Yaskawa INFORM job: X2_38-47,64(1)(90,180).JBI

/JOB
//NAME X2_38-47,64(1)(90,180)
//POS
///NPOS 477,477,477,26,0,0
///TOOL 0
///POSTYPE PULSE
///PULSE
C00000=10776,-116726,-133110,-1428,79202,-268
C00001=121301,-101656,-130574,15140,106953,26685
C00002=120740,-100574,-124017,14929,103680,26084
C00003=120691,-100743,-123189,14892,103111,25997
C00004=120691,-101012,-123023,14875,102879,25968
C00005=120694,-100727,-123199,14892,103125,25999
C00006=120263,-93974,-120700,15099,105066,26103
C00007=120694,-100727,-123199,14892,103125,25999
C00008=121303,-103883,-129892,15002,105440,26491
C00009=121309,-101301,-130428,15148,107041,26699
C00010=120755,-99767,-124232,14968,104207,26155
C00011=120700,-99774,-123449,14938,103747,26079
C00012=120700,-100712,-122892,14879,102948,25979
C00013=120685,-100384,-123078,14901,103225,26009
C00014=120255,-93653,-120581,15108,105156,26112
C00015=120685,-100384,-123078,14901,103225,26009
C00016=121293,-103472,-129753,15014,105563,26504
C00017=114791,-117911,-130965,19588,74628,29967
C00018=114769,-122713,-124135,20312,68344,28880
C00019=114477,-110584,-116158,20272,69659,29005
C00020=114421,-108517,-114081,20323,69469,28951
C00021=114421,-108669,-113508,20377,69064,28879
C00022=114502,-108614,-114130,20291,69431,28974
C00023=116741,-105993,-113204,19215,69642,29832
C00024=114502,-108614,-114130,20291,69431,28974
C00025=119599,-132627,-121815,19129,61042,29452
C00026=135151,-106131,-113172,10502,66286,36044
C00027=134382,-104032,-112419,10838,66989,35834
C00028=133562,-101757,-111587,11194,67742,35614
C00029=135151,-106131,-113172,10502,66286,36044
C00030=114538,-130880,-126635,20790,65904,28347
C00031=100256,-119338,-132400,19781,92736,-17009
C00032=115252,-134637,-128783,15911,82002,-19716
C00033=118597,-124593,-122817,15129,82811,-18454
C00034=119849,-120977,-120499,14834,83003,-18000
C00035=119848,-121103,-118880,14863,81976,-18124
C00036=119849,-120977,-120499,14834,83003,-18000
C00037=134184,-142802,-124917,2858,68148,-11180
C00038=133176,-135816,-122960,3144,70568,-11480
C00039=134184,-142802,-124917,2858,68148,-11180
C00040=110326,-92448,-108322,23569,98205,-21456
C00041=112623,-92143,-108201,23254,97666,-20755
C00042=110326,-92448,-108322,23569,98205,-21456
C00043=105090,-96290,-113946,24376,100996,-22735
C00044=105112,-88407,-119445,25319,107768,-21250
C00045=126458,-130213,-127441,-18734,86324,24062
C00046=122565,-122494,-122126,-18005,86127,22734
C00047=121090,-119592,-120022,-17718,85999,22241
C00048=121089,-119765,-118419,-17734,84972,22390
C00049=121090,-119592,-120022,-17718,85999,22241
C00050=121090,-119716,-118696,-17731,85160,22363
C00051=120619,-113401,-116618,-17615,86937,21943
C00052=121090,-119716,-118696,-17731,85160,22363
C00053=120691,-116357,-117549,-17638,86049,22096
C00054=118089,-117386,-117887,-17123,85200,21315
C00055=120691,-116357,-117549,-17638,86049,22096
C00056=125936,-126318,-124843,-18636,86589,23840
C00057=125953,-122568,-132013,-18690,92614,22924
C00058=117644,-124381,-130105,6983,115370,-67992
C00059=119593,-136528,-130318,6950,109138,-67660
C00060=120425,-140611,-129416,6959,106433,-67520
C00061=120425,-140322,-128375,6938,105944,-67549
C00062=120287,-139878,-129033,6943,106584,-67561
C00063=121808,-147552,-131144,7070,103828,-67181
C00064=120287,-139878,-129033,6943,106584,-67561
C00065=117523,-124132,-129146,6933,114921,-68065
C00066=117634,-108923,-132591,7489,118176,-67765
C00067=119077,-97405,-129626,2848,111310,-9091
C00068=112934,-122170,-124968,9693,82630,-11419
C00069=114889,-112052,-118675,9157,83718,-10686
C00070=115614,-108714,-115508,8968,83408,-10468
C00071=115614,-108962,-114752,8976,82823,-10510
C00072=115614,-108688,-115602,8966,83479,-10463
C00073=130338,-117040,-117457,-5173,77211,-4432
C00074=129550,-114521,-116623,-4914,77941,-4728
C00075=131152,-119600,-118288,-5441,76463,-4123
C00076=115450,-106601,-114144,9007,83670,-10503
C00077=117654,-103921,-113183,8408,84218,-9737
C00078=115450,-106601,-114144,9007,83670,-10503
C00079=112794,-119726,-122752,9732,82540,-11472
C00080=112816,-114614,-129461,9677,89201,-10949
C00081=124267,-125778,-125536,-12618,81617,14637
C00082=121749,-115664,-119377,-11934,82621,13684
C00083=120813,-112238,-116231,-11692,82317,13397
C00084=120812,-112414,-115451,-11705,81758,13450
C00085=120848,-112349,-116241,-11703,82272,13413
C00086=119586,-107060,-114409,-11339,83657,12862
C00087=120848,-112349,-116241,-11703,82272,13413
C00088=124307,-126037,-124767,-12644,81031,14711
C00089=124281,-122814,-131176,-12539,86499,14147
C00090=130647,-155525,-127944,-40400,54320,55258
C00091=124412,-146323,-123540,-36852,53123,52512
C00092=122059,-142698,-121760,-35413,52755,51453
C00093=119008,-142706,-121763,-33902,51510,50382
C00094=122059,-142698,-121760,-35413,52755,51453
C00095=119813,-142714,-121776,-34308,51836,50667
C00096=119829,-137326,-119074,-33845,52767,50322
C00097=119813,-142714,-121776,-34308,51836,50667
C00098=119893,-119020,-120433,-30427,61542,47434
C00099=120958,-113296,-116932,-30756,62602,47571
C00100=120971,-118070,-117370,-31352,60722,48150
C00101=120958,-113296,-116932,-30756,62602,47571
C00102=130647,-155525,-127944,-40400,54320,55258
C00103=121972,-140000,-127461,-3525,22047,40740
C00104=114503,-126631,-127045,28228,88345,28238
C00105=115418,-120062,-121213,28067,87856,28460
C00106=115767,-117777,-118144,28010,87108,28410
C00107=115767,-117863,-117333,28016,86625,28294
C00108=115798,-117876,-117463,28010,86680,28319
C00109=115506,-111666,-115391,28051,88476,28642
C00110=115798,-117876,-117463,28010,86680,28319
C00111=114535,-126949,-125608,28226,87406,28022
C00112=81132,-132100,-132064,22325,96940,18748
C00113=82014,-125321,-126186,22252,96583,18997
C00114=82351,-123063,-123074,22185,95795,18971
C00115=82354,-123167,-122323,22159,95314,18883
C00116=82329,-123147,-122467,22165,95412,18892
C00117=83163,-116500,-120334,22218,97147,19515
C00118=82329,-123147,-122467,22165,95412,18892
C00119=81992,-125617,-124767,22197,95637,18813
C00120=81110,-132470,-130662,22266,95968,18558
C00121=88413,-113418,-132573,32131,117765,52556
C00122=88284,-148255,-125485,32887,110398,70729
C00123=90408,-157751,-124889,32381,105124,70012
C00124=91344,-160468,-123864,32301,103041,69779
C00125=91347,-158891,-122215,32272,102866,69728
C00126=106792,-136481,-118062,29763,111204,74713
C00127=106248,-142899,-119829,29161,109458,74003
C00128=106792,-136481,-118062,29763,111204,74713
C00129=72811,-175927,-123443,35029,98716,64074
C00130=76149,-179694,-124176,35896,96158,64586
C00131=72811,-175927,-123443,35029,98716,64074
C00132=69241,-166504,-125806,34856,105362,64752
C00133=100814,-129767,-126176,13403,120642,68982
C00134=124653,-147507,-132240,-11278,113041,68250
C00135=122082,-159833,-132453,-11465,106593,67927
C00136=120953,-158348,-130532,-11731,106021,67572
C00137=120953,-156920,-128819,-11709,105706,67603
C00138=120952,-157581,-129221,-11703,105616,67612
C00139=120981,-170969,-132443,-11421,100817,68083
C00140=120958,-161991,-130311,-11601,104052,67766
C00141=120973,-170778,-133362,-11455,101467,68019
C00142=117530,-170630,-133328,-12326,101017,66845
C00143=120973,-170778,-133362,-11455,101467,68019
C00144=124784,-154865,-133680,-10989,110216,68576
C00145=122322,-137878,-131274,5971,121779,67906
C00146=120548,-145044,-127252,18536,119036,66813
C00147=120555,-156847,-127343,17506,113306,65855
C00148=120558,-160498,-126573,17182,111059,65507
C00149=120558,-158961,-124938,17154,110851,65476
C00150=120618,-159187,-125406,17199,111003,65522
C00151=120626,-166810,-127194,16864,108302,65121
C00152=120618,-159187,-125406,17199,111003,65522
C00153=120603,-144021,-125705,18473,118618,66761
C00154=115387,-132374,-123926,32562,106734,81694
C00155=118372,-141379,-123449,32107,101406,81342
C00156=119656,-144207,-122551,32012,99204,81226
C00157=119656,-143343,-121080,31963,98811,81114
C00158=119656,-144508,-123075,32029,99348,81268
C00159=131320,-114613,-113969,28597,111497,86004
C00160=131699,-120616,-115930,28265,109708,85685
C00161=131320,-114613,-113969,28597,111497,86004
C00162=105239,-169544,-124716,37289,88926,74807
C00163=108884,-170779,-124983,37802,86985,75650
C00164=105239,-169544,-124716,37289,88926,74807
C00165=99694,-161827,-127351,36723,95805,74832
C00166=131992,-100814,-126478,21663,116809,-46067
C00167=134007,-144842,-130967,18968,105768,-42043
C00168=134012,-143545,-127522,18820,104388,-42265
C00169=134287,-143929,-127856,18860,104334,-42172
C00170=133739,-135079,-123901,19000,106464,-42030
C00171=134883,-141438,-125704,18944,104153,-41980
C00172=134047,-144089,-127650,2764,111311,-58462
C00173=133934,-142264,-127061,2747,111888,-58492
C00174=135137,-137834,-120022,-13482,118747,-82298
C00175=135243,-139443,-120837,-14584,119263,-83981
C00176=134030,-142235,-124150,-15187,119626,-84533
C00177=119630,-122416,-133334,-16028,118546,-61096
C00178=134341,-125466,-134740,-10815,104436,-21672
C00179=120614,-100166,-121253,-7350,89365,11707
C00180=120622,-93660,-109595,-7359,85566,11930
C00181=122164,-90812,-108950,-7802,86761,12352
C00182=122198,-95853,-109304,-7828,84412,12509
C00183=122169,-92312,-107914,-7809,85365,12440
C00184=120622,-95353,-109162,-7367,84435,11995
C00185=122930,-76145,-100981,6392,88235,-3317
C00186=120621,-96600,-101892,16342,67221,-11741
C00187=120621,-96191,-103793,16192,68548,-11553
C00188=120639,-92247,-111396,15618,75005,-10677
C00189=188010,-107595,-125638,-17104,94805,24250
C00190=188020,-110122,-123495,-17031,92300,24603
C00191=185947,-121236,-125624,-16555,87669,24535
C00192=188801,-108952,-121724,-17183,91986,24909
C00193=188123,-110345,-123595,-17051,92269,24642
C00194=188114,-107825,-125741,-17124,94773,24289
C00195=177438,-122732,-133224,-14695,89877,21402
C00196=133569,-113989,-134534,-14289,94663,20149
C00197=119624,-110386,-135117,-7911,77851,79525
C00198=120615,-106635,-127104,-8473,74968,80030
C00199=127443,-106562,-124997,-15724,75089,81341
C00200=131001,-109651,-124953,-19889,73665,82237
C00201=120615,-106612,-127117,-8473,74988,80029
C00202=122620,-125184,-116655,-35316,53565,49443
C00203=120771,-121294,-114839,-33930,53551,48531
C00204=120821,-127755,-115028,-35341,50909,49582
C00205=120642,-147349,-113928,-41520,42291,53633
C00206=121034,-119467,-113769,-30359,65887,57979
C00207=122683,-120749,-115245,-30946,66698,58435
C00208=127694,-124296,-119025,-32687,68997,59841
C00209=127721,-118762,-131765,-31151,78153,27047
C00210=126237,-112945,-130032,-468,65797,4909
C00211=102361,-117345,-122757,6013,83638,-2551
C00212=102141,-118134,-119975,6094,81548,-2725
C00213=98567,-98899,-113703,7629,92375,-6440
C00214=118458,-104373,-115843,2992,90210,3061
C00215=122853,-105034,-115394,3962,88114,-4114
C00216=120609,-124185,-121101,4570,77097,-5239
C00217=120610,-123821,-123927,4542,79018,-5168
C00218=108948,-109237,-131335,7817,91844,-8301
C00219=115305,-101104,-129841,7326,117578,-44729
C00220=120606,-132359,-125648,5649,119733,-79611
C00221=120606,-131978,-122596,5547,118059,-79698
C00222=119593,-130601,-120983,5189,117844,-80105
C00223=120607,-131015,-120967,5517,117554,-79725
C00224=120606,-130958,-120980,5521,117590,-79725
C00225=120845,-129993,-119164,13944,117173,-67367
C00226=120606,-131851,-120987,13891,117375,-67436
C00227=120606,-132395,-123921,14113,118858,-67242
C00228=111305,-120759,-132293,17375,98141,-32748
C00229=120609,-124691,-119154,16638,71592,-14867
C00230=120609,-124440,-116582,16774,70197,-15066
C00231=120608,-124590,-115864,16826,69701,-15139
C00232=120609,-125347,-120005,-8811,76712,5958
C00233=120608,-124852,-119907,-8803,76903,5945
C00234=120384,-124859,-117862,-18190,76465,18975
C00235=120609,-124884,-118955,-18205,77141,18954
C00236=120609,-124961,-121688,-18108,78705,18718
C00237=132640,-106780,-128323,-23054,110263,-28369
C00238=120602,-139315,-124713,-24306,112781,-84362
C00239=120602,-138068,-121544,-24057,111582,-84094
C00240=120390,-136653,-120014,-24070,111324,-84123
C00241=111209,-136679,-122958,-3333,116425,-79190
C00242=120603,-138114,-123112,-90,115982,-75572
C00243=112873,-131131,-118331,19290,115700,-70424
C00244=107669,-134044,-117364,27346,113285,-69054
C00245=103576,-133216,-119553,26575,116197,-70036
C00246=103610,-135048,-130246,28186,121222,-68648
C00247=111190,-129681,-128447,36946,96833,-72948
C00248=111854,-129032,-128166,43025,93670,-81713
C00249=147502,-118658,-119533,35927,77679,-72524
C00250=147511,-119004,-116560,36172,76036,-73070
C00251=147515,-119022,-115332,36276,75411,-73279
C00252=147547,-116234,-125968,15022,114340,-70681
C00253=147515,-116012,-125840,15022,114380,-70688
C00254=147502,-115929,-125780,17177,108602,-60467
C00255=147494,-115895,-125723,16722,102508,-50684
C00256=147493,-115916,-125679,13964,96968,-41110
C00257=147497,-115970,-125656,10645,93613,-33926
C00258=147501,-116025,-125648,8199,92025,-29507
C00259=147506,-116072,-125646,5516,90867,-25066
C00260=147508,-116095,-125646,5516,90856,-25066
C00261=147505,-115163,-126691,5523,91973,-25018
C00262=147498,-112805,-128627,5545,94366,-24915
C00263=120610,-124729,-127429,-5691,77135,5542
C00264=120610,-125478,-124917,-5733,75213,5631
C00265=93121,-107602,-117934,17182,85224,-17308
C00266=100441,-109277,-120513,9088,85830,-5866
C00267=100640,-111519,-121837,6589,85674,558
C00268=115372,-129625,-126716,-4058,77034,4532
C00269=121142,-123508,-124723,-1462,78235,1570
C00270=113513,-125119,-124854,4552,77079,3092
C00271=116416,-125599,-125007,2130,76614,5633
C00272=113500,-125769,-125064,4555,76869,3083
C00273=117672,-122584,-124070,3211,77699,4516
C00274=120796,-120742,-123533,2204,78209,5572
C00275=125774,-129632,-127388,-3161,76112,11172
C00276=120611,-124694,-128184,-1477,78993,9385
C00277=-2000,-120083,-131752,-1890,40973,0
C00278=15972,-110889,-128286,10965,59905,43045
C00279=101389,-60822,-75148,-6919,68546,70102
C00280=115790,69230,64798,8053,66131,71909
C00281=120830,71540,61874,4756,55589,66514
C00282=120535,76858,72419,5134,51864,66212
C00283=120418,79487,77321,5314,50212,66075
C00284=120418,81305,81326,5435,48689,65991
C00285=120418,79487,77321,5314,50212,66075
C00286=121101,73566,71896,4942,50464,66384
C00287=120640,77942,77238,5256,49458,66131
C00288=121101,73566,71896,4942,50464,66384
C00289=121527,66226,57370,4418,55590,66797
C00290=120817,39260,26615,-5828,57686,79569
C00291=120487,42228,33767,-5849,54800,79594
C00292=120357,43570,36815,-5865,53609,79607
C00293=120357,44263,39245,-5952,52477,79673
C00294=120357,43570,36815,-5865,53609,79607
C00295=121171,39929,34748,-6347,53075,79981
C00296=120657,42834,37803,-6102,52651,79790
C00297=121171,39929,34748,-6347,53075,79981
C00298=121648,35573,24568,-6294,57116,79932
C00299=109578,65571,33028,8923,84264,70984
C00300=101389,-60822,-75148,-6919,68546,70102
C00301=96929,-90691,-89138,-5080,61517,23019
C00302=96929,-90691,-89138,-5080,61517,-27168
C00303=116056,-23990,-45922,-4976,84420,-46374
C00304=133997,38575,-5386,-4879,105902,-64390
C00305=134430,35731,-4221,-4855,103756,-64161
C00306=134605,34491,-3252,-4839,102536,-64054
C00307=134604,34193,-2477,-4825,101908,-64030
C00308=134605,34666,-3678,-4847,102887,-64068
C00309=133324,38381,1851,-4717,101326,-64430
C00310=133984,36157,-436,-4773,101627,-64224
C00311=133324,38381,1851,-4717,101326,-64430
C00312=132740,42105,45,-4739,104308,-64739
C00313=134038,40743,-3018,-12196,109842,-66951
C00314=134155,37294,-2552,-12029,107844,-66703
C00315=134216,35637,-2156,-11948,106779,-66572
C00316=134210,35418,-1183,-11898,106081,-66504
C00317=134138,36618,-275,-11900,106128,-66533
C00318=134308,36004,-906,-11910,106222,-66482
C00319=134138,36772,-681,-11923,106449,-66566
C00320=133552,41863,-495,-12102,108819,-67011
C00321=143157,-5596,-33734,-3459,84138,17748
C00322=146617,-6443,-23161,-4534,77380,19112
C00323=149281,-2495,-17370,-9500,77350,25048
C00324=149281,-2461,-16373,-9521,76762,25094
C00325=149281,-2503,-17669,-9494,77528,25035
C00326=148457,-726,-16200,-9269,77441,24757
C00327=149281,-2503,-17669,-9494,77528,25035
C00328=157589,4412,-9593,-22718,80450,41052
C00329=157226,5016,-8132,-22675,79802,41042
C00330=156592,4240,-8798,-22542,79640,40841
C00331=157226,4947,-9136,-22642,80340,40940
C00332=149281,-2387,-22338,-9412,80423,24814
C00333=149381,11612,-10676,-29411,77480,-58612
C00334=146879,26424,7173,-29053,73659,-58594
C00335=146667,27066,10077,-29192,72305,-58326
C00336=146666,27163,11157,-29282,71765,-58183
C00337=147639,24675,7343,-29416,73040,-58133
C00338=147917,24004,8167,-29618,72393,-57848
C00339=147086,25920,10012,-29396,71969,-58068
C00340=147917,24004,8167,-29618,72393,-57848
C00341=148686,22081,722,-29377,75807,-58446
C00342=135892,33292,-131,-24559,77407,-63614
C00343=147017,27605,-1759,-28452,79091,-59917
C00344=146805,27832,419,-28491,77938,-59710
C00345=146803,27699,1600,-28565,77235,-59535
C00346=147749,25558,-2150,-28746,78615,-59523
C00347=148390,24338,-1607,-29025,77984,-59121
C00348=147556,26192,183,-28786,77573,-59333
C00349=148390,24338,-1607,-29025,77984,-59121
C00350=149162,23542,-7999,-28991,81344,-59682
C00351=148025,26294,-7040,-28591,81698,-60189
C00352=147485,26714,-2602,-28593,79299,-59793
C00353=148219,27923,188,-28907,78577,-59336
C00354=148098,27627,1558,-28961,77659,-59149
C00355=147271,26975,-740,-28610,78335,-59633
C00356=147888,25428,-868,-28863,77908,-59292
C00357=147063,27300,949,-28626,77494,-59501
C00358=147888,25428,-868,-28863,77908,-59292
C00359=148652,24637,-7261,-28828,81272,-59852
C00360=129846,-17397,-52274,-16165,101048,-68229
C00361=103949,-6271,-30701,-7884,96105,-76175
C00362=94102,16895,-5866,-4380,94047,-79161
C00363=94024,14878,-3719,-4358,91692,-79105
C00364=93993,14152,-2780,-4351,90742,-79083
C00365=93993,14253,-1030,-4349,89719,-79047
C00366=93993,14152,-2780,-4351,90742,-79083
C00367=93685,20015,4382,-4321,89334,-79138
C00368=93881,17120,1686,-4338,89515,-79078
C00369=93685,20015,4382,-4321,89334,-79138
C00370=93796,22544,1176,-4343,92603,-79213
C00371=95224,-25687,-42365,-27028,60157,-72238
C00372=94111,-23276,-36997,-26973,57954,-72128
C00373=93676,-22234,-34203,-27071,56755,-71994
C00374=93677,-22196,-33100,-27266,56165,-71832
C00375=94095,-27015,-37738,-27384,56638,-71778
C00376=94165,-26445,-35973,-27662,55954,-71554
C00377=93910,-23559,-33944,-27450,56079,-71704
C00378=94165,-26445,-35973,-27662,55954,-71554
C00379=95768,-30118,-43626,-27714,58991,-71694
C00380=98687,-54699,-75805,-10421,73482,-70446
C00381=149776,12587,-27486,-12781,89603,18869
C00382=147726,21450,-15619,-10072,89467,18633
C00383=146063,28308,-6532,-8014,89346,18417
C00384=138620,21928,-10233,6772,82015,-93
C00385=138085,14099,-20532,6917,84360,-139
C00386=145828,23811,-13081,-8275,88592,27851
C00387=146877,26263,-7760,-8549,86699,28314
C00388=147056,24986,-14909,-8600,90423,28118
C00389=133623,24371,-15503,12505,92341,3955
C00390=141603,20096,-23343,-17631,90771,-45924
C00391=158767,23906,411,-41116,69770,-54212
C00392=157814,26218,6288,-41375,67476,-53693
C00393=157867,28101,9341,-41641,66811,-53385
C00394=155436,20095,3135,-35869,57411,-53274
C00395=154956,17275,-617,-35322,57921,-53695
C00396=155612,13879,-7263,-34858,60124,-54192
C00397=161259,32771,9254,-48678,77350,-54240
C00398=157220,20825,1180,-47844,74428,-54765
C00399=156964,21547,2982,-47923,73788,-54568
C00400=157920,25665,6992,-48239,74051,-54221
C00401=147580,194,-26885,-31933,72794,-56440
C00402=143572,-20191,-42827,-30403,70798,-57447
C00403=143289,15562,-12775,-40560,73024,-60435
C00404=161747,40468,15313,-46928,78664,-54425
C00405=163277,53845,31778,-50790,82736,-52233
C00406=162151,47089,24526,-50527,82761,-52828
C00407=160571,34350,9025,-46543,78569,-54946
C00408=152167,20307,-8359,-43656,76922,-58109
C00409=138097,34809,-8347,-11830,105930,-64747
C00410=138271,31970,-7074,-11701,103756,-64474
C00411=130058,42665,5328,-10329,107941,-67432
C00412=128254,38945,1428,-10381,108204,-68082
C00413=132059,42740,2082,-10449,110188,-66939
C00414=140613,2619,-37521,-15617,92132,-63158
C00415=170472,-48867,-31078,-12436,82300,-51309
C00416=161833,-30139,-32162,-12294,91042,-55174
C00417=111128,62365,52281,11955,55160,64549
C00418=111043,67239,62048,12539,51743,64100
C00419=108717,50085,54686,27686,34855,61667
C00420=111212,53885,58893,25958,33489,62752
C00421=111212,51875,53923,24699,35329,63437
C00422=113215,66301,56846,11015,54091,65302
C00423=121898,77388,65564,-1855,57299,70150
C00424=121470,82378,75801,-1732,53556,70040
C00425=123537,68913,65820,-7103,44835,71627
C00426=122634,66158,62455,-6429,45412,71158
C00427=121410,79209,71888,-1686,54335,70003
C00428=120651,73746,61164,-1269,58111,69644
C00429=113189,52303,49996,-7645,51731,77534
C00430=112734,56976,59397,-7777,48333,77603
C00431=115145,46398,55711,-16226,36410,80621
C00432=110709,39595,48522,-12260,36543,78075
C00433=109962,48589,50053,-6120,49525,76289
C00434=108655,45336,42401,-5185,52457,75559
C00435=161833,-30139,-32162,-12294,91042,-55174
C00436=151365,-63626,-36101,-12306,75003,-57224
C00437=105296,-38491,-50476,268,85780,-72725
C00438=93205,-23584,-36354,2491,84954,-76766
C00439=93975,-23467,-34641,2355,83937,-76526
C00440=95202,-23238,-34476,2131,83922,-76117
C00441=94250,-23197,-36080,2300,84954,-76417
C00442=93848,-22027,-39325,2370,87561,-76502
C00443=94651,-21766,-39138,-7100,89212,-77956
C00444=94455,-23170,-36061,-7070,86599,-77874
C00445=95552,-23013,-34317,-7248,85706,-77455
C00446=94465,-23468,-34640,-7076,85579,-77814
C00447=93466,-23543,-36325,-6911,86486,-78200
C00448=93670,-22147,-39411,-6941,89101,-78276
C00449=92980,-26767,-42567,-6357,64758,-77223
C00450=92830,-24983,-37315,-6405,62444,-77148
C00451=93722,-23870,-34926,-6909,61625,-76767
C00452=95877,-23183,-34437,-9028,62075,-75930
C00453=95090,-24132,-36711,-8569,62895,-76288
C00454=95328,-25868,-41938,-8524,65219,-76375
C00455=95261,-25907,-41974,-7480,65026,-76408
C00456=95085,-24145,-36729,-7536,62706,-76321
C00457=95607,-23367,-34574,-7858,61838,-76065
C00458=94456,-23753,-34846,-6874,61626,-76507
C00459=92783,-25001,-37319,-5340,62272,-77201
C00460=92870,-26808,-42587,-5281,64581,-77276
C00461=120452,-88146,-86102,-21652,66713,-67139
C00462=165262,-16782,-33522,-47685,80918,-53825
C00463=161018,-5245,-12472,-47809,73866,-52405
C00464=160660,-4212,-10170,-47919,73070,-52184
C00465=158378,-12349,-16601,-47497,71708,-52652
C00466=160281,-13132,-19159,-47644,73518,-52603
C00467=159752,-17175,-25374,-47188,74446,-53337
C00468=138959,36905,-6200,-11882,105806,-64445
C00469=139137,34092,-4934,-11755,103651,-64172
C00470=139758,34761,-2776,-11748,102772,-63879
C00471=136129,25909,-11433,-11506,103045,-65122
C00472=135629,25545,-13414,-11524,103991,-65380
C00473=138452,-5129,-43961,-15809,88138,-63518
C00474=104837,-81827,-69761,-4542,63447,-73998
C00475=84134,-123556,-96733,-5664,74963,-81774
C00476=10907,-117335,-90652,18762,63715,59495
BC00000=165804,522273,1075193
BC00001=35800,181198,1075139
BC00002=35800,181198,1075139
BC00003=35800,181198,1075139
BC00004=35800,181198,1075139
BC00005=35800,181198,1075139
BC00006=35800,181198,1075139
BC00007=35800,181198,1075139
BC00008=35800,181198,1075139
BC00009=81762,189115,1075139
BC00010=81762,189115,1075139
BC00011=81762,189115,1075139
BC00012=81762,189115,1075139
BC00013=81762,189115,1075139
BC00014=81762,189115,1075139
BC00015=81762,189115,1075139
BC00016=81762,189115,1075139
BC00017=183222,281904,1075139
BC00018=183222,281904,1075139
BC00019=183222,281904,1075139
BC00020=183222,281904,1075139
BC00021=183222,281904,1075139
BC00022=183222,281904,1075139
BC00023=183222,281904,1075139
BC00024=183222,281904,1075139
BC00025=183222,281904,1075139
BC00026=183222,281904,1075139
BC00027=183222,281904,1075139
BC00028=183222,281904,1075139
BC00029=183222,281904,1075139
BC00030=183222,281904,1075139
BC00031=277064,248649,1075139
BC00032=289773,243398,1075139
BC00033=289773,243398,1075139
BC00034=289773,243398,1075139
BC00035=289773,243398,1075139
BC00036=289773,243398,1075139
BC00037=289773,243398,1075139
BC00038=289773,243398,1075139
BC00039=289773,243398,1075139
BC00040=289773,243398,1075139
BC00041=289773,243398,1075139
BC00042=289773,243398,1075139
BC00043=289773,243398,1075139
BC00044=289773,243398,1075139
BC00045=261284,244615,1075139
BC00046=261284,244615,1075139
BC00047=261284,244615,1075139
BC00048=261284,244615,1075139
BC00049=261284,244615,1075139
BC00050=261284,244615,1075139
BC00051=261284,244615,1075139
BC00052=261284,244615,1075139
BC00053=261284,244615,1075139
BC00054=261284,244615,1075139
BC00055=261284,244615,1075139
BC00056=261284,244615,1075139
BC00057=261284,244615,1075139
BC00058=293731,217262,1075139
BC00059=293731,217262,1075139
BC00060=293731,217262,1075139
BC00061=293731,217262,1075139
BC00062=293731,217262,1075139
BC00063=293731,217262,1075139
BC00064=293731,217262,1075139
BC00065=293731,217262,1075139
BC00066=293731,232104,1075139
BC00067=262313,306825,1075139
BC00068=265671,329387,1075139
BC00069=265671,329387,1075139
BC00070=265671,329387,1075139
BC00071=265671,329387,1075139
BC00072=265671,329387,1075139
BC00073=265671,329387,1075139
BC00074=265671,329387,1075139
BC00075=265671,329387,1075139
BC00076=265671,329387,1075139
BC00077=265671,329387,1075139
BC00078=265671,329387,1075139
BC00079=265671,329387,1075139
BC00080=265671,329387,1075139
BC00081=272036,349446,1075139
BC00082=272036,349446,1075139
BC00083=272036,349446,1075139
BC00084=272036,349446,1075139
BC00085=272036,349446,1075139
BC00086=272036,349446,1075139
BC00087=272036,349446,1075139
BC00088=272036,349446,1075139
BC00089=272036,349446,1075139
BC00090=294062,256541,1075139
BC00091=294062,256541,1075139
BC00092=294062,256541,1075139
BC00093=294062,256541,1075139
BC00094=294062,256541,1075139
BC00095=294062,256541,1075139
BC00096=294062,256541,1075139
BC00097=294062,256541,1075139
BC00098=294062,256541,1075139
BC00099=294062,256541,1075139
BC00100=294062,256541,1075139
BC00101=294062,256541,1075139
BC00102=294062,256541,1075139
BC00103=349994,338464,1075139
BC00104=398158,240026,1075139
BC00105=398158,240026,1075139
BC00106=398158,240026,1075139
BC00107=398158,240026,1075139
BC00108=398158,240026,1075139
BC00109=398158,240026,1075139
BC00110=398158,240026,1075139
BC00111=398158,240026,1075139
BC00112=398158,236035,1075139
BC00113=398158,236035,1075139
BC00114=398158,236035,1075139
BC00115=398158,236035,1075139
BC00116=398158,236035,1075139
BC00117=398158,236035,1075139
BC00118=398158,236035,1075139
BC00119=398158,236035,1075139
BC00120=398158,236035,1075139
BC00121=398158,319428,1075139
BC00122=398158,372381,1075139
BC00123=398158,372381,1075139
BC00124=398158,372381,1075139
BC00125=398158,372381,1075139
BC00126=398158,372381,1075139
BC00127=398158,372381,1075139
BC00128=398158,372381,1075139
BC00129=398158,372381,1075139
BC00130=398158,372381,1075139
BC00131=398158,372381,1075139
BC00132=398158,372381,1075139
BC00133=396432,362940,1075139
BC00134=394806,360489,1075139
BC00135=394806,360489,1075139
BC00136=394806,360489,1075139
BC00137=394806,360489,1075139
BC00138=394806,360489,1075139
BC00139=394806,360489,1075139
BC00140=394806,360489,1075139
BC00141=394806,360489,1075139
BC00142=394806,360489,1075139
BC00143=394806,360489,1075139
BC00144=394806,360489,1075139
BC00145=355367,356213,1075139
BC00146=324584,345067,1075139
BC00147=324584,345067,1075139
BC00148=324584,345067,1075139
BC00149=324584,345067,1075139
BC00150=324584,345067,1075139
BC00151=324584,345067,1075139
BC00152=324584,345067,1075139
BC00153=324584,345067,1075139
BC00154=311925,382226,1075139
BC00155=311925,382226,1075139
BC00156=311925,382226,1075139
BC00157=311925,382226,1075139
BC00158=311925,382226,1075139
BC00159=311925,382226,1075139
BC00160=311925,382226,1075139
BC00161=311925,382226,1075139
BC00162=311925,382226,1075139
BC00163=311925,382226,1075139
BC00164=311925,382226,1075139
BC00165=311925,382226,1075139
BC00166=316265,227195,1075139
BC00167=312557,199845,1075139
BC00168=307887,202335,1075139
BC00169=306018,203331,1075139
BC00170=306018,203331,1075139
BC00171=306018,203331,1075139
BC00172=283244,197415,1075139
BC00173=316914,216368,1075139
BC00174=284717,205535,1075136
BC00175=281628,202596,1075139
BC00176=279091,197007,1075139
BC00177=280135,229568,1075139
BC00178=281301,312859,1075139
BC00179=282622,370317,1075139
BC00180=284842,365275,1075139
BC00181=285731,363258,1075139
BC00182=285731,363258,1075139
BC00183=285731,363258,1075139
BC00184=239170,337138,1075139
BC00185=271891,349841,1075139
BC00186=285584,357140,1075139
BC00187=288450,363211,1075139
BC00188=288450,363211,1075139
BC00189=136038,186132,1075139
BC00190=136333,180752,1075139
BC00191=136451,178600,1075139
BC00192=86038,169868,1075139
BC00193=85456,171940,1075139
BC00194=85161,177320,1075139
BC00195=85161,322446,1075139
BC00196=394559,334508,1075139
BC00197=335349,251306,1075139
BC00198=336692,255151,1075139
BC00199=337229,254342,1075139
BC00200=337252,247401,1075139
BC00201=336714,248211,1075139
BC00202=295924,262948,1075139
BC00203=295924,262948,1075139
BC00204=295924,262948,1075139
BC00205=295924,262948,1075139
BC00206=295924,262948,1075139
BC00207=295924,262948,1075139
BC00208=295924,262948,1075139
BC00209=295924,262948,1075139
BC00210=393665,278082,1075139
BC00211=398158,268381,1075139
BC00212=398158,263147,1075139
BC00213=398158,261489,1075139
BC00214=364745,251487,1075139
BC00215=369183,252743,1075139
BC00216=369626,254869,1075139
BC00217=370734,260182,1075139
BC00218=370734,341715,1075139
BC00219=340677,355670,1075139
BC00220=313124,360643,1075139
BC00221=312412,366022,1075139
BC00222=312128,368174,1075139
BC00223=307349,368159,1075139
BC00224=268099,368041,1075136
BC00225=280159,368452,1075139
BC00226=281255,366425,1075139
BC00227=283995,361357,1075139
BC00228=290712,292171,1075139
BC00229=293746,260926,1075139
BC00230=290432,255685,1075139
BC00231=289106,253589,1075139
BC00232=241713,247157,1075139
BC00233=279816,253757,1075139
BC00234=264120,250428,1075139
BC00235=262531,252178,1075139
BC00236=258558,256552,1075139
BC00237=314933,317196,1075139
BC00238=378455,362215,1075139
BC00239=380899,367360,1075139
BC00240=381877,369418,1075139
BC00241=398158,364218,1075139
BC00242=361433,364075,1075139
BC00243=386371,371318,1075139
BC00244=398158,372977,1075139
BC00245=398158,368566,1075139
BC00246=398158,368566,1075139
BC00247=256476,224361,1075139
BC00248=237908,188682,1075139
BC00249=237908,174656,1075139
BC00250=232917,176445,1075139
BC00251=230921,177160,1075139
BC00252=178443,139274,1075139
BC00253=212997,158656,1075139
BC00254=227025,169975,1075139
BC00255=235497,185625,1075139
BC00256=237112,203182,1075139
BC00257=233250,216751,1075139
BC00258=228038,225928,1075139
BC00259=223162,232173,1075139
BC00260=220666,234564,1075139
BC00261=222327,235432,1075139
BC00262=225648,237168,1075139
BC00263=141832,275443,1075139
BC00264=143112,269810,1075139
BC00265=143623,267556,1075139
BC00266=137635,265405,1075139
BC00267=129678,262548,1075139
BC00268=134104,259263,1075139
BC00269=148655,263166,1075139
BC00270=116922,247641,1075139
BC00271=115677,247045,1075139
BC00272=111398,244993,1075139
BC00273=111398,244993,1075139
BC00274=111398,244993,1075139
BC00275=110907,247158,1075139
BC00276=109924,251488,1075139
BC00277=131733,514405,1075139
BC00278=21198,517278,429866
BC00279=66799,465991,419725
BC00280=110224,417152,337633
BC00281=136713,400556,283945
BC00282=136713,400556,283945
BC00283=136713,400556,283945
BC00284=136713,400556,283945
BC00285=136713,400556,283945
BC00286=136713,400556,283945
BC00287=136713,400556,283945
BC00288=136713,400556,283945
BC00289=136713,400556,283945
BC00290=163178,400556,279134
BC00291=163178,400556,279134
BC00292=163178,400556,279134
BC00293=163178,400556,279134
BC00294=163178,400556,279134
BC00295=163178,400556,279134
BC00296=163178,400556,279134
BC00297=163178,400556,279134
BC00298=163178,400556,279134
BC00299=110224,417152,230098
BC00300=66799,465991,419725
BC00301=66799,545915,419725
BC00302=252749,519251,169722
BC00303=278530,473105,170836
BC00304=322792,429821,131675
BC00305=322792,429821,131675
BC00306=322792,429821,131675
BC00307=322792,429821,131675
BC00308=322792,429821,131675
BC00309=322792,429821,131675
BC00310=322792,429821,131675
BC00311=322792,429821,131675
BC00312=322792,429821,131675
BC00313=340391,437456,125654
BC00314=340391,437456,125654
BC00315=340391,437456,125654
BC00316=340391,437456,125654
BC00317=340391,437456,125654
BC00318=340391,437456,125654
BC00319=340391,437456,125654
BC00320=340391,437456,125654
BC00321=309461,406297,200874
BC00322=309461,406297,200874
BC00323=309461,406297,200874
BC00324=309461,406297,200874
BC00325=309461,406297,200874
BC00326=309461,406297,200874
BC00327=309461,406297,200874
BC00328=309461,406297,200874
BC00329=309461,406297,200874
BC00330=309461,406297,200874
BC00331=309461,406297,200874
BC00332=309461,406297,200874
BC00333=303662,400556,204886
BC00334=303662,415917,204886
BC00335=303662,415917,204886
BC00336=303662,415917,204886
BC00337=303662,415917,204886
BC00338=303662,415917,204886
BC00339=303662,415917,204886
BC00340=303662,415917,204886
BC00341=303662,415917,204886
BC00342=312134,452819,139026
BC00343=343990,437458,139026
BC00344=343990,437458,139026
BC00345=343990,437458,139026
BC00346=343990,437458,139026
BC00347=343990,437458,139026
BC00348=343990,437458,139026
BC00349=343990,437458,139026
BC00350=343990,437458,139026
BC00351=374473,456471,136048
BC00352=374473,456471,136048
BC00353=374473,456471,136048
BC00354=374473,456471,136048
BC00355=374473,456471,136048
BC00356=374473,456471,136048
BC00357=374473,456471,136048
BC00358=374473,456471,136048
BC00359=374473,456471,136048
BC00360=300917,439314,218872
BC00361=283877,440048,250459
BC00362=276304,440374,264498
BC00363=276304,440374,264498
BC00364=276304,440374,264498
BC00365=276304,440374,264498
BC00366=276304,440374,264498
BC00367=276304,440374,264498
BC00368=276304,440374,264498
BC00369=276304,440374,264498
BC00370=276304,440374,264498
BC00371=248841,426339,138655
BC00372=248841,426339,138655
BC00373=248841,426339,138655
BC00374=248841,426339,138655
BC00375=248841,426339,138655
BC00376=248841,426339,138655
BC00377=248841,426339,138655
BC00378=248841,426339,138655
BC00379=248841,426339,138655
BC00380=248841,426339,138655
BC00381=315035,431339,94305
BC00382=315035,431339,94305
BC00383=315035,431339,94305
BC00384=315035,431339,94305
BC00385=315035,431339,94305
BC00386=315035,431339,94305
BC00387=315035,431339,94305
BC00388=315035,431339,94305
BC00389=315035,431339,94305
BC00390=315035,431339,94305
BC00391=334446,428157,129137
BC00392=334446,428157,129137
BC00393=334446,428157,129137
BC00394=334446,428157,129137
BC00395=334446,428157,129137
BC00396=334446,428157,129137
BC00397=313795,418314,120096
BC00398=302567,411800,120096
BC00399=302567,411800,120096
BC00400=302567,411800,120096
BC00401=302567,411800,120096
BC00402=302567,411800,120096
BC00403=334446,460819,94191
BC00404=398158,460819,94191
BC00405=398158,460819,94191
BC00406=398158,460819,94191
BC00407=398158,460819,94191
BC00408=366302,460819,94191
BC00409=350696,437944,121163
BC00410=350696,437944,121163
BC00411=326438,437944,121163
BC00412=326438,437944,121163
BC00413=326438,437944,121163
BC00414=326438,437944,121163
BC00415=382552,521140,422200
BC00416=167327,521140,639421
BC00417=112225,400556,268007
BC00418=112225,400556,268007
BC00419=112225,400556,268007
BC00420=112225,400556,268007
BC00421=112225,400556,268007
BC00422=112225,400556,268007
BC00423=121098,400556,252431
BC00424=121098,400556,252431
BC00425=121098,400556,252431
BC00426=121098,400556,252431
BC00427=121098,400556,252431
BC00428=121098,400556,252431
BC00429=121321,400556,329672
BC00430=121321,400556,329672
BC00431=121321,400556,329672
BC00432=121321,400556,329672
BC00433=121321,400556,329672
BC00434=121321,400556,329672
BC00435=167327,521140,639421
BC00436=323590,521140,422200
BC00437=275640,416909,237205
BC00438=299235,416909,237205
BC00439=299235,416909,237205
BC00440=299235,416909,237205
BC00441=299235,416909,237205
BC00442=299235,416909,237205
BC00443=279462,405807,237631
BC00444=279462,405807,237631
BC00445=279462,405807,237631
BC00446=279462,405807,237631
BC00447=279462,405807,237631
BC00448=279462,405807,237631
BC00449=280262,429298,181651
BC00450=280262,429298,181651
BC00451=280262,429298,181651
BC00452=280262,429298,181651
BC00453=280262,429298,181651
BC00454=280262,429298,181651
BC00455=277533,427766,181657
BC00456=277533,427766,181657
BC00457=277533,427766,181657
BC00458=277533,427766,181657
BC00459=277533,427766,181657
BC00460=277533,427766,181657
BC00461=297259,418542,184288
BC00462=335725,400556,189417
BC00463=335725,400556,189417
BC00464=335725,400556,189417
BC00465=335725,400556,189417
BC00466=335725,400556,189417
BC00467=335725,400556,189417
BC00468=319519,421779,121460
BC00469=319519,421779,121460
BC00470=319519,421779,121460
BC00471=319519,421779,121460
BC00472=319519,421779,121460
BC00473=319519,421779,121460
BC00474=252021,473498,250459
BC00475=250740,505808,243879
BC00476=165804,522273,534000
EC00000=-798156,-1296783
EC00001=-798156,-1296783
EC00002=-798156,-1296783
EC00003=-798156,-1296783
EC00004=-798156,-1296783
EC00005=-798156,-1296783
EC00006=-798156,-1296783
EC00007=-798156,-1296783
EC00008=-798156,-1296783
EC00009=-798156,-1296783
EC00010=-798156,-1296783
EC00011=-798156,-1296783
EC00012=-798156,-1296783
EC00013=-798156,-1296783
EC00014=-798156,-1296783
EC00015=-798156,-1296783
EC00016=-798156,-1296783
EC00017=-798156,-1296783
EC00018=-798156,-1296783
EC00019=-798156,-1296783
EC00020=-798156,-1296783
EC00021=-798156,-1296783
EC00022=-798156,-1296783
EC00023=-798156,-1296783
EC00024=-798156,-1296783
EC00025=-798156,-1296783
EC00026=-798156,-1296783
EC00027=-798156,-1296783
EC00028=-798156,-1296783
EC00029=-798156,-1296783
EC00030=-798156,-1296783
EC00031=-798156,-1296783
EC00032=-798156,-1296783
EC00033=-798156,-1296783
EC00034=-798156,-1296783
EC00035=-798156,-1296783
EC00036=-798156,-1296783
EC00037=-798156,-1296783
EC00038=-798156,-1296783
EC00039=-798156,-1296783
EC00040=-798156,-1296783
EC00041=-798156,-1296783
EC00042=-798156,-1296783
EC00043=-798156,-1296783
EC00044=-798156,-1296783
EC00045=-798156,-1296783
EC00046=-798156,-1296783
EC00047=-798156,-1296783
EC00048=-798156,-1296783
EC00049=-798156,-1296783
EC00050=-798156,-1296783
EC00051=-798156,-1296783
EC00052=-798156,-1296783
EC00053=-798156,-1296783
EC00054=-798156,-1296783
EC00055=-798156,-1296783
EC00056=-798156,-1296783
EC00057=-798156,-1296783
EC00058=-798156,-1296783
EC00059=-798156,-1296783
EC00060=-798156,-1296783
EC00061=-798156,-1296783
EC00062=-798156,-1296783
EC00063=-798156,-1296783
EC00064=-798156,-1296783
EC00065=-798156,-1296783
EC00066=-798156,-1296783
EC00067=-798156,-1296783
EC00068=-798156,-1296783
EC00069=-798156,-1296783
EC00070=-798156,-1296783
EC00071=-798156,-1296783
EC00072=-798156,-1296783
EC00073=-798156,-1296783
EC00074=-798156,-1296783
EC00075=-798156,-1296783
EC00076=-798156,-1296783
EC00077=-798156,-1296783
EC00078=-798156,-1296783
EC00079=-798156,-1296783
EC00080=-798156,-1296783
EC00081=-798156,-1296783
EC00082=-798156,-1296783
EC00083=-798156,-1296783
EC00084=-798156,-1296783
EC00085=-798156,-1296783
EC00086=-798156,-1296783
EC00087=-798156,-1296783
EC00088=-798156,-1296783
EC00089=-798156,-1296783
EC00090=-798156,-1296783
EC00091=-798156,-1296783
EC00092=-798156,-1296783
EC00093=-798156,-1296783
EC00094=-798156,-1296783
EC00095=-798156,-1296783
EC00096=-798156,-1296783
EC00097=-798156,-1296783
EC00098=-798156,-1296783
EC00099=-798156,-1296783
EC00100=-798156,-1296783
EC00101=-798156,-1296783
EC00102=-798156,-1296783
EC00103=-798156,-1296783
EC00104=-798156,-1296783
EC00105=-798156,-1296783
EC00106=-798156,-1296783
EC00107=-798156,-1296783
EC00108=-798156,-1296783
EC00109=-798156,-1296783
EC00110=-798156,-1296783
EC00111=-798156,-1296783
EC00112=-798156,-1296783
EC00113=-798156,-1296783
EC00114=-798156,-1296783
EC00115=-798156,-1296783
EC00116=-798156,-1296783
EC00117=-798156,-1296783
EC00118=-798156,-1296783
EC00119=-798156,-1296783
EC00120=-798156,-1296783
EC00121=-798156,-1296783
EC00122=-798156,-1296783
EC00123=-798156,-1296783
EC00124=-798156,-1296783
EC00125=-798156,-1296783
EC00126=-798156,-1296783
EC00127=-798156,-1296783
EC00128=-798156,-1296783
EC00129=-798156,-1296783
EC00130=-798156,-1296783
EC00131=-798156,-1296783
EC00132=-798156,-1296783
EC00133=-798156,-1296783
EC00134=-798156,-1296783
EC00135=-798156,-1296783
EC00136=-798156,-1296783
EC00137=-798156,-1296783
EC00138=-798156,-1296783
EC00139=-798156,-1296783
EC00140=-798156,-1296783
EC00141=-798156,-1296783
EC00142=-798156,-1296783
EC00143=-798156,-1296783
EC00144=-798156,-1296783
EC00145=-798156,-1296783
EC00146=-798156,-1296783
EC00147=-798156,-1296783
EC00148=-798156,-1296783
EC00149=-798156,-1296783
EC00150=-798156,-1296783
EC00151=-798156,-1296783
EC00152=-798156,-1296783
EC00153=-798156,-1296783
EC00154=-798156,-1296783
EC00155=-798156,-1296783
EC00156=-798156,-1296783
EC00157=-798156,-1296783
EC00158=-798156,-1296783
EC00159=-798156,-1296783
EC00160=-798156,-1296783
EC00161=-798156,-1296783
EC00162=-798156,-1296783
EC00163=-798156,-1296783
EC00164=-798156,-1296783
EC00165=-798156,-1296783
EC00166=-798156,-1296783
EC00167=-798156,-1296783
EC00168=-798156,-1296783
EC00169=-798156,-1296783
EC00170=-798156,-1296783
EC00171=-798156,-1296783
EC00172=-798156,-1296783
EC00173=-798156,-1296783
EC00174=-798155,-1296782
EC00175=-798156,-1296783
EC00176=-798156,-1296783
EC00177=-798156,-1296783
EC00178=-798156,-1296783
EC00179=-798156,-1296783
EC00180=-798156,-1296783
EC00181=-798156,-1296783
EC00182=-798156,-1296783
EC00183=-798156,-1296783
EC00184=-798156,-1296783
EC00185=-798156,-1296783
EC00186=-798156,-1296783
EC00187=-798156,-1296783
EC00188=-798156,-1296783
EC00189=-798156,-1296783
EC00190=-798156,-1296783
EC00191=-798156,-1296783
EC00192=-798156,-1296783
EC00193=-798156,-1296783
EC00194=-798156,-1296783
EC00195=-798156,-1296783
EC00196=-798156,-1296783
EC00197=-798156,-1296783
EC00198=-798156,-1296783
EC00199=-798156,-1296783
EC00200=-798156,-1296783
EC00201=-798156,-1296783
EC00202=-798156,-1296783
EC00203=-798156,-1296783
EC00204=-798156,-1296783
EC00205=-798156,-1296783
EC00206=-798156,-1296783
EC00207=-798156,-1296783
EC00208=-798156,-1296783
EC00209=-798156,-1296783
EC00210=-798156,-1296783
EC00211=-798156,-1296783
EC00212=-798156,-1296783
EC00213=-798156,-1296783
EC00214=-798156,-1296783
EC00215=-798155,-1296782
EC00216=-798156,-1296783
EC00217=-798156,-1296783
EC00218=-798156,-1296783
EC00219=-798156,-1296783
EC00220=-798156,-1296783
EC00221=-798156,-1296783
EC00222=-798156,-1296783
EC00223=-798156,-1296783
EC00224=-798155,-1296782
EC00225=-798156,-1296783
EC00226=-798156,-1296783
EC00227=-798156,-1296783
EC00228=-798156,-1296783
EC00229=-798156,-1296783
EC00230=-798156,-1296783
EC00231=-798156,-1296783
EC00232=-798156,-1296783
EC00233=-798156,-1296783
EC00234=-798156,-1296783
EC00235=-798156,-1296783
EC00236=-798156,-1296783
EC00237=-798156,-1296783
EC00238=-798156,-1296783
EC00239=-798156,-1296783
EC00240=-798156,-1296783
EC00241=-798156,-1296783
EC00242=-798156,-1296783
EC00243=-798156,-1296783
EC00244=-798156,-1296783
EC00245=-798156,-1296783
EC00246=-798156,-1296783
EC00247=-798156,-1296783
EC00248=-798156,-1296783
EC00249=-798156,-1296783
EC00250=-798156,-1296783
EC00251=-798156,-1296783
EC00252=-798156,-1296783
EC00253=-798156,-1296783
EC00254=-798156,-1296783
EC00255=-798156,-1296783
EC00256=-798156,-1296783
EC00257=-798156,-1296783
EC00258=-798156,-1296783
EC00259=-798156,-1296783
EC00260=-798156,-1296783
EC00261=-798156,-1296783
EC00262=-798156,-1296783
EC00263=-798156,-1296783
EC00264=-798156,-1296783
EC00265=-798156,-1296783
EC00266=-798156,-1296783
EC00267=-798156,-1296783
EC00268=-798156,-1296783
EC00269=-798156,-1296783
EC00270=-798156,-1296783
EC00271=-798156,-1296783
EC00272=-798156,-1296783
EC00273=-798156,-1296783
EC00274=-798156,-1296783
EC00275=-798156,-1296783
EC00276=-798156,-1296783
EC00277=-798156,-1296783
EC00278=-798156,-1296783
EC00279=-798156,-1296783
EC00280=-798156,-1296783
EC00281=-798156,-1296783
EC00282=-798156,-1296783
EC00283=-798156,-1296783
EC00284=-798156,-1296783
EC00285=-798156,-1296783
EC00286=-798156,-1296783
EC00287=-798156,-1296783
EC00288=-798156,-1296783
EC00289=-798156,-1296783
EC00290=-798156,-1296783
EC00291=-798156,-1296783
EC00292=-798156,-1296783
EC00293=-798156,-1296783
EC00294=-798156,-1296783
EC00295=-798156,-1296783
EC00296=-798156,-1296783
EC00297=-798156,-1296783
EC00298=-798156,-1296783
EC00299=-798156,-1296783
EC00300=-798156,-1296783
EC00301=-798156,-1296783
EC00302=-798156,-1296783
EC00303=-798156,-1296783
EC00304=-798156,-1296783
EC00305=-798156,-1296783
EC00306=-798156,-1296783
EC00307=-798156,-1296783
EC00308=-798156,-1296783
EC00309=-798156,-1296783
EC00310=-798156,-1296783
EC00311=-798156,-1296783
EC00312=-798156,-1296783
EC00313=-798156,-1296783
EC00314=-798156,-1296783
EC00315=-798156,-1296783
EC00316=-798156,-1296783
EC00317=-798156,-1296783
EC00318=-798156,-1296783
EC00319=-798156,-1296783
EC00320=-798156,-1296783
EC00321=-798156,-1296783
EC00322=-798156,-1296783
EC00323=-798156,-1296783
EC00324=-798156,-1296783
EC00325=-798156,-1296783
EC00326=-798156,-1296783
EC00327=-798156,-1296783
EC00328=-798156,-1296783
EC00329=-798156,-1296783
EC00330=-798156,-1296783
EC00331=-798156,-1296783
EC00332=-798156,-1296783
EC00333=-798156,-1296783
EC00334=-798156,-1296783
EC00335=-798156,-1296783
EC00336=-798156,-1296783
EC00337=-798156,-1296783
EC00338=-798156,-1296783
EC00339=-798156,-1296783
EC00340=-798156,-1296783
EC00341=-798156,-1296783
EC00342=-798156,-1296783
EC00343=-798156,-1296783
EC00344=-798156,-1296783
EC00345=-798156,-1296783
EC00346=-798156,-1296783
EC00347=-798156,-1296783
EC00348=-798156,-1296783
EC00349=-798156,-1296783
EC00350=-798156,-1296783
EC00351=-798156,-1296783
EC00352=-798156,-1296783
EC00353=-798156,-1296783
EC00354=-798156,-1296783
EC00355=-798156,-1296783
EC00356=-798156,-1296783
EC00357=-798156,-1296783
EC00358=-798156,-1296783
EC00359=-798156,-1296783
EC00360=-798156,-1296783
EC00361=-798156,-1296783
EC00362=-798156,-1296783
EC00363=-798156,-1296783
EC00364=-798156,-1296783
EC00365=-798156,-1296783
EC00366=-798156,-1296783
EC00367=-798156,-1296783
EC00368=-798156,-1296783
EC00369=-798156,-1296783
EC00370=-798156,-1296783
EC00371=-798156,-1296783
EC00372=-798156,-1296783
EC00373=-798156,-1296783
EC00374=-798156,-1296783
EC00375=-798156,-1296783
EC00376=-798156,-1296783
EC00377=-798156,-1296783
EC00378=-798156,-1296783
EC00379=-798156,-1296783
EC00380=-798156,-1296783
EC00381=-798156,-1296783
EC00382=-798156,-1296783
EC00383=-798156,-1296783
EC00384=-798156,-1296783
EC00385=-798156,-1296783
EC00386=-798156,-1296783
EC00387=-798156,-1296783
EC00388=-798156,-1296783
EC00389=-798156,-1296783
EC00390=-798156,-1296783
EC00391=-798156,-1296783
EC00392=-798156,-1296783
EC00393=-798156,-1296783
EC00394=-798156,-1296783
EC00395=-798156,-1296783
EC00396=-798156,-1296783
EC00397=-798156,-1296783
EC00398=-798156,-1296783
EC00399=-798156,-1296783
EC00400=-798156,-1296783
EC00401=-798156,-1296783
EC00402=-798156,-1296783
EC00403=-798156,-1296783
EC00404=-798156,-1296783
EC00405=-798156,-1296783
EC00406=-798156,-1296783
EC00407=-798156,-1296783
EC00408=-798156,-1296783
EC00409=-798156,-1296783
EC00410=-798156,-1296783
EC00411=-798156,-1296783
EC00412=-798156,-1296783
EC00413=-798156,-1296783
EC00414=-798156,-1296783
EC00415=-798156,-1296783
EC00416=-798156,-1296783
EC00417=-798156,-1296783
EC00418=-798156,-1296783
EC00419=-798156,-1296783
EC00420=-798156,-1296783
EC00421=-798156,-1296783
EC00422=-798156,-1296783
EC00423=-798156,-1296783
EC00424=-798156,-1296783
EC00425=-798156,-1296783
EC00426=-798156,-1296783
EC00427=-798156,-1296783
EC00428=-798156,-1296783
EC00429=-798156,-1296783
EC00430=-798156,-1296783
EC00431=-798156,-1296783
EC00432=-798156,-1296783
EC00433=-798156,-1296783
EC00434=-798156,-1296783
EC00435=-798156,-1296783
EC00436=-798156,-1296783
EC00437=-798156,-1296783
EC00438=-798156,-1296783
EC00439=-798156,-1296783
EC00440=-798156,-1296783
EC00441=-798156,-1296783
EC00442=-798156,-1296783
EC00443=-798156,-1296783
EC00444=-798156,-1296783
EC00445=-798156,-1296783
EC00446=-798156,-1296783
EC00447=-798156,-1296783
EC00448=-798156,-1296783
EC00449=-798156,-1296783
EC00450=-798156,-1296783
EC00451=-798156,-1296783
EC00452=-798156,-1296783
EC00453=-798156,-1296783
EC00454=-798156,-1296783
EC00455=-798156,-1296783
EC00456=-798156,-1296783
EC00457=-798156,-1296783
EC00458=-798156,-1296783
EC00459=-798156,-1296783
EC00460=-798156,-1296783
EC00461=-798156,-1296783
EC00462=-798156,-1296783
EC00463=-798156,-1296783
EC00464=-798156,-1296783
EC00465=-798156,-1296783
EC00466=-798156,-1296783
EC00467=-798156,-1296783
EC00468=-798156,-1296783
EC00469=-798156,-1296783
EC00470=-798156,-1296783
EC00471=-798156,-1296783
EC00472=-798156,-1296783
EC00473=-798156,-1296783
EC00474=-798156,-1296783
EC00475=-798156,-1296783
EC00476=-798156,-1296783
///POSTYPE BASE
///RECTAN
///RCONF 0,0,0,0,1,0,0,0,0,0,0,0,0,0,0,0,0,0,0,0,0,0,0,0
P00006=2.006,1.622,-0.565,0.0000,0.0000,0.0000
P00021=0.073,2.058,-0.109,0.0000,0.0000,0.0000
P00022=2.006,1.622,-0.565,0.0000,0.0000,0.0000
///RCONF 0,0,0,0,0,0,0,0,0,0,0,0,0,0,0,0,0,0,0,0,0,0,0,0
P00023=-2.957,-4.083,2.762,0.0000,0.0000,0.0000
P00024=-1.466,-0.226,-0.419,0.0000,0.0000,0.0000
P00025=3.643,0.007,-2.585,0.0000,0.0000,0.0000
P00026=2.644,0.055,-2.583,0.0000,0.0000,0.0000
P00027=2.278,0.099,-4.210,0.0000,0.0000,0.0000
P00028=-1.778,-0.182,-2.050,0.0000,0.0000,0.0000
P00029=1.749,4.006,-0.261,0.0000,0.0000,0.0000
P00030=-0.014,-0.768,0.131,0.0000,0.0000,0.0000
P00031=-0.170,0.039,-0.647,0.0000,0.0000,0.0000
P00032=-0.423,0.157,3.222,0.0000,0.0000,0.0000
P00033=0.854,-1.099,3.047,0.0000,0.0000,0.0000
///RCONF 0,0,0,0,1,0,0,0,0,0,0,0,0,0,0,0,0,0,0,0,0,0,0,0
P00034=-8.151,9.743,-4.393,0.0000,0.0000,0.0000
///RCONF 0,0,0,0,0,0,0,0,0,0,0,0,0,0,0,0,0,0,0,0,0,0,0,0
P00042=-0.220,0.371,-0.613,0.0000,0.0000,0.0000
P00043=-0.179,-5.890,-3.227,0.0000,0.0000,0.0000
P00044=-8.560,-7.557,-5.232,0.0000,0.0000,0.0000
P00045=-8.836,-6.632,-1.438,0.0000,0.0000,0.0000
P00046=-7.725,-0.107,-2.878,0.0000,0.0000,0.0000
///RCONF 0,1,0,0,0,0,0,0,0,0,0,0,0,0,0,0,0,0,0,0,0,0,0,0
P00047=0.052,4.745,-6.175,0.0000,0.0000,0.0000
///RCONF 0,0,0,0,0,0,0,0,0,0,0,0,0,0,0,0,0,0,0,0,0,0,0,0
P00048=-10.315,0.035,-3.101,0.0000,0.0000,0.0000
P00049=-9.638,1.690,-2.627,0.0000,0.0000,0.0000
P00050=-0.123,2.174,-1.314,0.0000,0.0000,0.0000
P00051=-5.945,4.696,-10.293,0.0000,0.0000,0.0000
P00060=1524.284,698.404,-261.973,-0.4635,36.8346,-1.2388
//INST
///DATE 2024/12/18 16:17
///ATTR SC,RW
///GROUP1 RB1,BS1
///GROUP2 ST1
NOP
'X2_38-47,64(1)(90,180)
'Down
MOVJ C00000 BC00000 VJ=100.00  +MOVJ EC00000 VJ=100.00
'Up
'Path S3659
SFTOF3D
MOVJ C00001 BC00001 VJ=100.00  +MOVJ EC00001 VJ=100.00
MOVL C00002 BC00002 V=666.7  +MOVJ EC00002 VJ=100.00
SMOVL C00003 BC00003 V=166.7  +MOVJ EC00003
SREFP 3 C00004 BC00004  +REFP EC00004
CALL JOB:SEARCH-R1-S13D
SET P021 P006
SFTON3D P021
SMOVL C00005 BC00005 V=166.7  +MOVJ EC00005
SREFP 3 C00006 BC00006  +REFP EC00006
CALL JOB:SEARCH-R1-S13D
SET P021 P006
SFTON3D P021
SMOVL C00007 BC00007 V=166.7  +MOVJ EC00007
MOVL C00008 BC00008 V=1000.0  +MOVJ EC00008 VJ=100.00
'EndPath S3659
'Path S4334
SFTOF3D
MOVJ C00009 BC00009 VJ=100.00  +MOVJ EC00009 VJ=100.00
MOVL C00010 BC00010 V=666.7  +MOVJ EC00010 VJ=100.00
SMOVL C00011 BC00011 V=166.7  +MOVJ EC00011
SREFP 3 C00012 BC00012  +REFP EC00012
CALL JOB:SEARCH-R1-S13D
SET P022 P006
SFTON3D P022
SMOVL C00013 BC00013 V=166.7  +MOVJ EC00013
SREFP 3 C00014 BC00014  +REFP EC00014
CALL JOB:SEARCH-R1-S13D
SET P022 P006
SFTON3D P022
SMOVL C00015 BC00015 V=166.7  +MOVJ EC00015
MOVL C00016 BC00016 V=1000.0  +MOVJ EC00016 VJ=100.00
'EndPath S4334
'Path S3657
SFTOF3D
MOVJ C00017 BC00017 VJ=100.00  +MOVJ EC00017 VJ=100.00
MOVJ C00018 BC00018 VJ=100.00  +MOVJ EC00018 VJ=100.00
MOVL C00019 BC00019 V=666.7  +MOVJ EC00019 VJ=100.00
SMOVL C00020 BC00020 V=166.7  +MOVJ EC00020
SREFP 3 C00021 BC00021  +REFP EC00021
CALL JOB:SEARCH-R1-S13D
SET P023 P006
SFTON3D P023
SMOVL C00022 BC00022 V=166.7  +MOVJ EC00022
SREFP 3 C00023 BC00023  +REFP EC00023
CALL JOB:SEARCH-R1-S13D
SET P023 P006
SFTON3D P023
SMOVL C00024 BC00024 V=166.7  +MOVJ EC00024
SMOVL C00025 BC00025 V=500.0  +MOVJ EC00025
SMOVL C00026 BC00026 V=800.0  +MOVJ EC00026
SMOVL C00027 BC00027 V=166.7  +MOVJ EC00027
SREFP 3 C00028 BC00028  +REFP EC00028
CALL JOB:SEARCH-R1-S13D
SET P023 P006
SFTON3D P023
SMOVL C00029 BC00029 V=250.0  +MOVJ EC00029
MOVL C00030 BC00030 V=1000.0  +MOVJ EC00030 VJ=100.00
'EndPath S3657
MOVJ C00031 BC00031 VJ=100.00  +MOVJ EC00031 VJ=100.00
'Path S3665
SFTOF3D
MOVJ C00032 BC00032 VJ=100.00  +MOVJ EC00032 VJ=100.00
MOVL C00033 BC00033 V=800.0  +MOVJ EC00033 VJ=100.00
SMOVL C00034 BC00034 V=166.7  +MOVJ EC00034
SREFP 3 C00035 BC00035  +REFP EC00035
CALL JOB:SEARCH-R1-S13D
SET P024 P006
SFTON3D P024
SMOVL C00036 BC00036 V=166.7  +MOVJ EC00036
SMOVL C00037 BC00037 V=166.7  +MOVJ EC00037
SREFP 3 C00038 BC00038  +REFP EC00038
CALL JOB:SEARCH-R1-S13D
SET P024 P006
SFTON3D P024
SMOVL C00039 BC00039 V=166.7  +MOVJ EC00039
SMOVL C00040 BC00040 V=166.7  +MOVJ EC00040
SREFP 3 C00041 BC00041  +REFP EC00041
CALL JOB:SEARCH-R1-S13D
SET P024 P006
SFTON3D P024
SMOVL C00042 BC00042 V=166.7  +MOVJ EC00042
MOVL C00043 BC00043 V=1000.0  +MOVJ EC00043 VJ=100.00
MOVL C00044 BC00044 V=1000.0  +MOVJ EC00044 VJ=100.00
'EndPath S3665
'Path S4335
SFTOF3D
MOVJ C00045 BC00045 VJ=100.00  +MOVJ EC00045 VJ=100.00
MOVL C00046 BC00046 V=800.0  +MOVJ EC00046 VJ=100.00
SMOVL C00047 BC00047 V=166.7  +MOVJ EC00047
SREFP 3 C00048 BC00048  +REFP EC00048
CALL JOB:SEARCH-R1-S13D
SET P025 P006
SFTON3D P025
SMOVL C00049 BC00049 V=166.7  +MOVJ EC00049
SMOVL C00050 BC00050 V=166.7  +MOVJ EC00050
SREFP 3 C00051 BC00051  +REFP EC00051
CALL JOB:SEARCH-R1-S13D
SET P025 P006
SFTON3D P025
SMOVL C00052 BC00052 V=166.7  +MOVJ EC00052
SMOVL C00053 BC00053 V=166.7  +MOVJ EC00053
SREFP 3 C00054 BC00054  +REFP EC00054
CALL JOB:SEARCH-R1-S13D
SET P025 P006
SFTON3D P025
SMOVL C00055 BC00055 V=166.7  +MOVJ EC00055
MOVL C00056 BC00056 V=1000.0  +MOVJ EC00056 VJ=100.00
MOVL C00057 BC00057 V=1000.0  +MOVJ EC00057 VJ=100.00
'EndPath S4335
'Path S3666
SFTOF3D
MOVJ C00058 BC00058 VJ=100.00  +MOVJ EC00058 VJ=100.00
MOVL C00059 BC00059 V=800.0  +MOVJ EC00059 VJ=100.00
SMOVL C00060 BC00060 V=166.7  +MOVJ EC00060
SREFP 3 C00061 BC00061  +REFP EC00061
CALL JOB:SEARCH-R1-S13D
SET P026 P006
SFTON3D P026
SMOVL C00062 BC00062 V=166.7  +MOVJ EC00062
SREFP 3 C00063 BC00063  +REFP EC00063
CALL JOB:SEARCH-R1-S13D
SET P026 P006
SFTON3D P026
SMOVL C00064 BC00064 V=166.7  +MOVJ EC00064
MOVL C00065 BC00065 V=1000.0  +MOVJ EC00065 VJ=100.00
'EndPath S3666
MOVJ C00066 BC00066 VJ=100.00  +MOVJ EC00066 VJ=100.00
MOVJ C00067 BC00067 VJ=100.00  +MOVJ EC00067 VJ=100.00
'Path S3661
SFTOF3D
MOVJ C00068 BC00068 VJ=100.00  +MOVJ EC00068 VJ=100.00
MOVL C00069 BC00069 V=800.0  +MOVJ EC00069 VJ=100.00
SMOVL C00070 BC00070 V=166.7  +MOVJ EC00070
SREFP 3 C00071 BC00071  +REFP EC00071
CALL JOB:SEARCH-R1-S13D
SET P027 P006
SFTON3D P027
SMOVL C00072 BC00072 V=166.7  +MOVJ EC00072
SMOVL C00073 BC00073 V=166.7  +MOVJ EC00073
SREFP 3 C00074 BC00074  +REFP EC00074
CALL JOB:SEARCH-R1-S13D
SET P027 P006
SFTON3D P027
SMOVL C00075 BC00075 V=250.0  +MOVJ EC00075
SMOVL C00076 BC00076 V=166.7  +MOVJ EC00076
SREFP 3 C00077 BC00077  +REFP EC00077
CALL JOB:SEARCH-R1-S13D
SET P027 P006
SFTON3D P027
SMOVL C00078 BC00078 V=166.7  +MOVJ EC00078
MOVL C00079 BC00079 V=1000.0  +MOVJ EC00079 VJ=100.00
MOVL C00080 BC00080 V=1000.0  +MOVJ EC00080 VJ=100.00
'EndPath S3661
'Path S4336
SFTOF3D
MOVJ C00081 BC00081 VJ=100.00  +MOVJ EC00081 VJ=100.00
MOVL C00082 BC00082 V=800.0  +MOVJ EC00082 VJ=100.00
SMOVL C00083 BC00083 V=166.7  +MOVJ EC00083
SREFP 3 C00084 BC00084  +REFP EC00084
CALL JOB:SEARCH-R1-S13D
SET P028 P006
SFTON3D P028
SMOVL C00085 BC00085 V=166.7  +MOVJ EC00085
SREFP 3 C00086 BC00086  +REFP EC00086
CALL JOB:SEARCH-R1-S13D
SET P028 P006
SFTON3D P028
SMOVL C00087 BC00087 V=166.7  +MOVJ EC00087
MOVL C00088 BC00088 V=1000.0  +MOVJ EC00088 VJ=100.00
'EndPath S4336
MOVJ C00089 BC00089 VJ=100.00  +MOVJ EC00089 VJ=100.00
'Path S4879
SFTOF3D
MOVJ C00090 BC00090 VJ=100.00  +MOVJ EC00090 VJ=100.00
MOVL C00091 BC00091 V=800.0  +MOVJ EC00091 VJ=100.00
SMOVL C00092 BC00092 V=166.7  +MOVJ EC00092
SREFP 3 C00093 BC00093  +REFP EC00093
CALL JOB:SEARCH-R1-S13D
SET P060 P006
SFTON3D P060
SMOVL C00094 BC00094 V=166.7  +MOVJ EC00094
SMOVL C00095 BC00095 V=166.7  +MOVJ EC00095
SREFP 3 C00096 BC00096  +REFP EC00096
CALL JOB:SEARCH-R1-S13D
SET P060 P006
SFTON3D P060
SMOVL C00097 BC00097 V=166.7  +MOVJ EC00097
SMOVL C00098 BC00098 V=250.0  +MOVJ EC00098
SMOVL C00099 BC00099 V=166.7  +MOVJ EC00099
SREFP 3 C00100 BC00100  +REFP EC00100
CALL JOB:SEARCH-R1-S13D
SET P060 P006
SFTON3D P060
SMOVL C00101 BC00101 V=166.7  +MOVJ EC00101
MOVL C00102 BC00102 V=1000.0  +MOVJ EC00102 VJ=100.00
'EndPath S4879
MOVJ C00103 BC00103 VJ=100.00  +MOVJ EC00103 VJ=100.00
'Path S3664
SFTOF3D
MOVJ C00104 BC00104 VJ=100.00  +MOVJ EC00104 VJ=100.00
MOVL C00105 BC00105 V=800.0  +MOVJ EC00105 VJ=100.00
SMOVL C00106 BC00106 V=166.7  +MOVJ EC00106
SREFP 3 C00107 BC00107  +REFP EC00107
CALL JOB:SEARCH-R1-S13D
SET P029 P006
SFTON3D P029
SMOVL C00108 BC00108 V=166.7  +MOVJ EC00108
SREFP 3 C00109 BC00109  +REFP EC00109
CALL JOB:SEARCH-R1-S13D
SET P029 P006
SFTON3D P029
SMOVL C00110 BC00110 V=166.7  +MOVJ EC00110
MOVL C00111 BC00111 V=1000.0  +MOVJ EC00111 VJ=100.00
'EndPath S3664
'Path S4337
SFTOF3D
MOVJ C00112 BC00112 VJ=100.00  +MOVJ EC00112 VJ=100.00
MOVL C00113 BC00113 V=800.0  +MOVJ EC00113 VJ=100.00
SMOVL C00114 BC00114 V=166.7  +MOVJ EC00114
SREFP 3 C00115 BC00115  +REFP EC00115
CALL JOB:SEARCH-R1-S13D
SET P030 P006
SFTON3D P030
SMOVL C00116 BC00116 V=166.7  +MOVJ EC00116
SREFP 3 C00117 BC00117  +REFP EC00117
CALL JOB:SEARCH-R1-S13D
SET P030 P006
SFTON3D P030
SMOVL C00118 BC00118 V=166.7  +MOVJ EC00118
MOVL C00119 BC00119 V=800.0  +MOVJ EC00119 VJ=100.00
MOVL C00120 BC00120 V=1000.0  +MOVJ EC00120 VJ=100.00
'EndPath S4337
MOVJ C00121 BC00121 VJ=100.00  +MOVJ EC00121 VJ=100.00
'Path S3663
SFTOF3D
MOVJ C00122 BC00122 VJ=100.00  +MOVJ EC00122 VJ=100.00
MOVL C00123 BC00123 V=800.0  +MOVJ EC00123 VJ=100.00
SMOVL C00124 BC00124 V=166.7  +MOVJ EC00124
SREFP 3 C00125 BC00125  +REFP EC00125
CALL JOB:SEARCH-R1-S13D
SET P031 P006
SFTON3D P031
SMOVL C00126 BC00126 V=166.7  +MOVJ EC00126
SREFP 3 C00127 BC00127  +REFP EC00127
CALL JOB:SEARCH-R1-S13D
SET P031 P006
SFTON3D P031
SMOVL C00128 BC00128 V=166.7  +MOVJ EC00128
SMOVL C00129 BC00129 V=166.7  +MOVJ EC00129
SREFP 3 C00130 BC00130  +REFP EC00130
CALL JOB:SEARCH-R1-S13D
SET P031 P006
SFTON3D P031
SMOVL C00131 BC00131 V=166.7  +MOVJ EC00131
MOVL C00132 BC00132 V=1000.0  +MOVJ EC00132 VJ=100.00
'EndPath S3663
MOVJ C00133 BC00133 VJ=100.00  +MOVJ EC00133 VJ=100.00
'Path S4338
SFTOF3D
MOVJ C00134 BC00134 VJ=100.00  +MOVJ EC00134 VJ=100.00
MOVL C00135 BC00135 V=800.0  +MOVJ EC00135 VJ=100.00
SMOVL C00136 BC00136 V=166.7  +MOVJ EC00136
SREFP 3 C00137 BC00137  +REFP EC00137
CALL JOB:SEARCH-R1-S13D
SET P032 P006
SFTON3D P032
SMOVL C00138 BC00138 V=166.7  +MOVJ EC00138
SREFP 3 C00139 BC00139  +REFP EC00139
CALL JOB:SEARCH-R1-S13D
SET P032 P006
SFTON3D P032
SMOVL C00140 BC00140 V=166.7  +MOVJ EC00140
SMOVL C00141 BC00141 V=166.7  +MOVJ EC00141
SREFP 3 C00142 BC00142  +REFP EC00142
CALL JOB:SEARCH-R1-S13D
SET P032 P006
SFTON3D P032
SMOVL C00143 BC00143 V=166.7  +MOVJ EC00143
MOVL C00144 BC00144 V=1000.0  +MOVJ EC00144 VJ=100.00
'EndPath S4338
MOVJ C00145 BC00145 VJ=100.00  +MOVJ EC00145 VJ=100.00
'Path S3662
SFTOF3D
MOVJ C00146 BC00146 VJ=100.00  +MOVJ EC00146 VJ=100.00
MOVL C00147 BC00147 V=800.0  +MOVJ EC00147 VJ=100.00
SMOVL C00148 BC00148 V=166.7  +MOVJ EC00148
SREFP 3 C00149 BC00149  +REFP EC00149
CALL JOB:SEARCH-R1-S13D
SET P033 P006
SFTON3D P033
SMOVL C00150 BC00150 V=166.7  +MOVJ EC00150
SREFP 3 C00151 BC00151  +REFP EC00151
CALL JOB:SEARCH-R1-S13D
SET P033 P006
SFTON3D P033
SMOVL C00152 BC00152 V=166.7  +MOVJ EC00152
MOVL C00153 BC00153 V=1000.0  +MOVJ EC00153 VJ=100.00
'EndPath S3662
'Path S4339
SFTOF3D
MOVJ C00154 BC00154 VJ=100.00  +MOVJ EC00154 VJ=100.00
MOVL C00155 BC00155 V=800.0  +MOVJ EC00155 VJ=100.00
SMOVL C00156 BC00156 V=166.7  +MOVJ EC00156
SREFP 3 C00157 BC00157  +REFP EC00157
CALL JOB:SEARCH-R1-S13D
SET P034 P006
SFTON3D P034
SMOVL C00158 BC00158 V=166.7  +MOVJ EC00158
SMOVL C00159 BC00159 V=166.7  +MOVJ EC00159
SREFP 3 C00160 BC00160  +REFP EC00160
CALL JOB:SEARCH-R1-S13D
SET P034 P006
SFTON3D P034
SMOVL C00161 BC00161 V=166.7  +MOVJ EC00161
SMOVL C00162 BC00162 V=166.7  +MOVJ EC00162
SREFP 3 C00163 BC00163  +REFP EC00163
CALL JOB:SEARCH-R1-S13D
SET P034 P006
SFTON3D P034
SMOVL C00164 BC00164 V=166.7  +MOVJ EC00164
MOVL C00165 BC00165 V=1000.0  +MOVJ EC00165 VJ=100.00
'EndPath S4339
MOVJ C00166 BC00166 VJ=100.00  +MOVJ EC00166 VJ=100.00
'Path W3667
SFTOF3D
SFTON3D P026
MOVJ C00167 BC00167 VJ=100.00  +MOVJ EC00167 VJ=100.00
SMOVL C00168 BC00168 V=800.0  +MOVJ EC00168
SREFP 1 C00169 BC00169  +REFP EC00169
SREFP 2 C00170 BC00170  +REFP EC00170
SMOVL C00171 BC00171 V=166.7 PL=0  +MOVJ EC00171
MACRO1 MJ#(0) ARGF21
ARCON
SWVON WEV#(100)
SMOVL C00172 BC00172 V=9.2  +MOVJ EC00172
SMOVL C00173 BC00173 V=9.2  +MOVJ EC00173
SMOVL C00174 BC00174 V=9.2  +MOVJ EC00174
ARCOF
SWVOF
SMOVL C00175 BC00175 V=800.0  +MOVJ EC00175
SMOVL C00176 BC00176 V=1000.0  +MOVJ EC00176
SFTOF3D
'EndPath W3667
MOVJ C00177 BC00177 VJ=100.00  +MOVJ EC00177 VJ=100.00
MOVJ C00178 BC00178 VJ=100.00  +MOVJ EC00178 VJ=100.00
'Path W3668
SSFTOF
SFTOF3D
SFTON3D P028
MOVJ C00179 BC00179 VJ=100.00  +MOVJ EC00179 VJ=100.00
SMOVL C00180 BC00180 V=800.0  +MOVJ EC00180
SREFP 1 C00181 BC00181  +REFP EC00181
SREFP 2 C00182 BC00182  +REFP EC00182
SMOVL C00183 BC00183 V=150.0 PL=0  +MOVJ EC00183
ARCON
SWVON WEV#(100)
SFTON3D P027
SMOVL C00184 BC00184 V=9.2  +MOVJ EC00184
SMOVL C00185 BC00185 V=9.2  +MOVJ EC00185
ARCOF
SWVOF
SMOVL C00186 BC00186 V=800.0  +MOVJ EC00186
SMOVL C00187 BC00187 V=1000.0  +MOVJ EC00187
SFTOF3D
'EndPath W3668
MOVJ C00188 BC00188 VJ=100.00  +MOVJ EC00188 VJ=100.00
'Path W4546
SFTOF3D
SFTON3D P022
MOVJ C00189 BC00189 VJ=100.00  +MOVJ EC00189 VJ=100.00
SMOVL C00190 BC00190 V=800.0  +MOVJ EC00190
SMOVL C00191 BC00191 V=150.0 PL=0  +MOVJ EC00191
MACRO1 MJ#(0) ARGF9
ARCON
SWVON WEV#(10)
SFTON3D P021
SMOVL C00192 BC00192 V=10.0  +MOVJ EC00192
ARCOF
SWVOF
SMOVL C00193 BC00193 V=800.0  +MOVJ EC00193
SMOVL C00194 BC00194 V=1000.0  +MOVJ EC00194
SFTOF3D
'EndPath W4546
'Path W4901
SFTOF3D
SFTON3D P060
MOVJ C00195 BC00195 VJ=100.00  +MOVJ EC00195 VJ=100.00
MOVJ C00196 BC00196 VJ=100.00  +MOVJ EC00196 VJ=100.00
MOVJ C00197 BC00197 VJ=100.00  +MOVJ EC00197 VJ=100.00
SMOVL C00198 BC00198 V=800.0  +MOVJ EC00198
SMOVL C00199 BC00199 V=150.0 PL=0  +MOVJ EC00199
MACRO1 MJ#(0) ARGF14
ARCON
SMOVL C00200 BC00200 V=10.8  +MOVJ EC00200
ARCOF
SMOVL C00201 BC00201 V=800.0  +MOVJ EC00201
SFTOF3D
'EndPath W4901
'Path W4880
SFTOF3D
SFTON3D P060
SMOVL C00202 BC00202 V=800.0  +MOVJ EC00202
SMOVL C00203 BC00203 V=150.0 PL=0  +MOVJ EC00203
ARCON
SMOVL C00204 BC00204 V=10.0  +MOVJ EC00204
SMOVL C00205 BC00205 V=10.0  +MOVJ EC00205
SMOVL C00206 BC00206 V=10.0  +MOVJ EC00206
ARCOF
SMOVL C00207 BC00207 V=800.0  +MOVJ EC00207
SMOVL C00208 BC00208 V=1000.0  +MOVJ EC00208
SFTOF3D
'EndPath W4880
MOVJ C00209 BC00209 VJ=100.00  +MOVJ EC00209 VJ=100.00
MOVJ C00210 BC00210 VJ=100.00  +MOVJ EC00210 VJ=100.00
'Path W4548
SFTOF3D
SFTON3D P030
MOVJ C00211 BC00211 VJ=100.00  +MOVJ EC00211 VJ=100.00
SMOVL C00212 BC00212 V=800.0  +MOVJ EC00212
SMOVL C00213 BC00213 V=150.0 PL=0  +MOVJ EC00213
MACRO1 MJ#(0) ARGF9
ARCON
SFTON3D P029
SMOVL C00214 BC00214 V=10.0  +MOVJ EC00214
SMOVL C00215 BC00215 V=10.0  +MOVJ EC00215
ARCOF
SMOVL C00216 BC00216 V=800.0  +MOVJ EC00216
SMOVL C00217 BC00217 V=1000.0  +MOVJ EC00217
SFTOF3D
'EndPath W4548
MOVJ C00218 BC00218 VJ=100.00  +MOVJ EC00218 VJ=100.00
MOVJ C00219 BC00219 VJ=100.00  +MOVJ EC00219 VJ=100.00
'Path W3671
SFTOF3D
SFTON3D P033
MOVJ C00220 BC00220 VJ=100.00  +MOVJ EC00220 VJ=100.00
SMOVL C00221 BC00221 V=800.0  +MOVJ EC00221
SMOVL C00222 BC00222 V=166.7 PL=0  +MOVJ EC00222
MACRO1 MJ#(0) ARGF14
ARCON
SMOVL C00223 BC00223 V=9.2  +MOVJ EC00223
SFTON3D P034
SMOVL C00224 BC00224 V=9.2  +MOVJ EC00224
SMOVL C00225 BC00225 V=9.2  +MOVJ EC00225
ARCOF
SMOVL C00226 BC00226 V=800.0  +MOVJ EC00226
SMOVL C00227 BC00227 V=1000.0  +MOVJ EC00227
SFTOF3D
'EndPath W3671
MOVJ C00228 BC00228 VJ=100.00  +MOVJ EC00228 VJ=100.00
'Path W3672
SFTOF3D
SFTON3D P024
MOVJ C00229 BC00229 VJ=100.00  +MOVJ EC00229 VJ=100.00
SMOVL C00230 BC00230 V=800.0  +MOVJ EC00230
SMOVL C00231 BC00231 V=166.7 PL=0  +MOVJ EC00231
ARCON
SMOVL C00232 BC00232 V=9.2  +MOVJ EC00232
SFTON3D P025
SMOVL C00233 BC00233 V=9.2  +MOVJ EC00233
SMOVL C00234 BC00234 V=9.2  +MOVJ EC00234
ARCOF
SMOVL C00235 BC00235 V=800.0  +MOVJ EC00235
SMOVL C00236 BC00236 V=1000.0  +MOVJ EC00236
SFTOF3D
'EndPath W3672
MOVJ C00237 BC00237 VJ=100.00  +MOVJ EC00237 VJ=100.00
'Path W3673
SFTOF3D
SFTON3D P032
MOVJ C00238 BC00238 VJ=100.00  +MOVJ EC00238 VJ=100.00
SMOVL C00239 BC00239 V=800.0  +MOVJ EC00239
SMOVL C00240 BC00240 V=166.7 PL=0  +MOVJ EC00240
ARCON
SMOVL C00241 BC00241 V=9.2  +MOVJ EC00241
SFTON3D P031
SMOVL C00242 BC00242 V=9.2  +MOVJ EC00242
SMOVL C00243 BC00243 V=9.2  +MOVJ EC00243
ARCOF
SMOVL C00244 BC00244 V=800.0  +MOVJ EC00244
SMOVL C00245 BC00245 V=1000.0  +MOVJ EC00245
SFTOF3D
'EndPath W3673
MOVJ C00246 BC00246 VJ=100.00  +MOVJ EC00246 VJ=100.00
'
MOVJ C00247 BC00247 VJ=100.00  +MOVJ EC00247 VJ=100.00
JUMP *VV
MOVJ C00248 BC00248 VJ=100.00  +MOVJ EC00248 VJ=100.00
'Path W3680
SFTOF3D
SFTON3D P023
MOVJ C00249 BC00249 VJ=100.00  +MOVJ EC00249 VJ=100.00
SMOVL C00250 BC00250 V=800.0  +MOVJ EC00250
SMOVL C00251 BC00251 V=166.7 PL=0  +MOVJ EC00251
SMOVL C00252 BC00252 V=10.0  +MOVJ EC00252
SMOVL C00253 BC00253 V=33.3  +MOVJ EC00253
SMOVL C00254 BC00254 V=33.3  +MOVJ EC00254
SMOVL C00255 BC00255 V=33.3  +MOVJ EC00255
SMOVL C00256 BC00256 V=10.0  +MOVJ EC00256
SMOVL C00257 BC00257 V=10.0  +MOVJ EC00257
SMOVL C00258 BC00258 V=10.0  +MOVJ EC00258
SMOVL C00259 BC00259 V=10.0  +MOVJ EC00259
SMOVL C00260 BC00260 V=10.0  +MOVJ EC00260
ARCOF
SMOVL C00261 BC00261 V=800.0  +MOVJ EC00261
SMOVL C00262 BC00262 V=1000.0  +MOVJ EC00262
SFTOF3D
'EndPath W3680
'Path W3681
*VV
SFTOF3D
SFTON3D P023
MOVJ C00263 BC00263 VJ=100.00  +MOVJ EC00263 VJ=100.00
SMOVL C00264 BC00264 V=800.0  +MOVJ EC00264
SMOVL C00265 BC00265 V=150.0 PL=0  +MOVJ EC00265
MACRO1 MJ#(0) ARGF9
ARCON
SMOVL C00266 BC00266 V=8.3  +MOVJ EC00266
SMOVL C00267 BC00267 V=8.3  +MOVJ EC00267
SMOVL C00268 BC00268 V=8.3  +MOVJ EC00268
SMOVL C00269 BC00269 V=8.3  +MOVJ EC00269
SMOVL C00270 BC00270 V=8.3  +MOVJ EC00270
SMOVL C00271 BC00271 V=8.3  +MOVJ EC00271
SMOVL C00272 BC00272 V=8.3  +MOVJ EC00272
SMOVL C00273 BC00273 V=8.3  +MOVJ EC00273
SMOVL C00274 BC00274 V=8.3  +MOVJ EC00274
ARCOF
SMOVL C00275 BC00275 V=800.0  +MOVJ EC00275
SMOVL C00276 BC00276 V=1000.0  +MOVJ EC00276
SFTOF3D
'EndPath W3681
'Down
MOVJ C00277 BC00277 VJ=100.00  +MOVJ EC00277 VJ=100.00
CALL JOB:CLEAN-R1_KM_NEW
'1
MOVJ C00278 BC00278 VJ=100.00  +MOVJ EC00278 VJ=100.00
MOVJ C00279 BC00279 VJ=100.00  +MOVJ EC00279 VJ=100.00
MOVJ C00280 BC00280 VJ=100.00  +MOVJ EC00280 VJ=100.00
'Path S4334
SFTOF3D
MOVJ C00281 BC00281 VJ=100.00  +MOVJ EC00281 VJ=100.00
MOVL C00282 BC00282 V=800.0  +MOVJ EC00282 VJ=100.00
SMOVL C00283 BC00283 V=166.7  +MOVJ EC00283
SREFP 3 C00284 BC00284  +REFP EC00284
CALL JOB:SEARCH-R1-S13D
SET P048 P006
SFTON3D P048
SMOVL C00285 BC00285 V=166.7  +MOVJ EC00285
SMOVL C00286 BC00286 V=166.7  +MOVJ EC00286
SREFP 3 C00287 BC00287  +REFP EC00287
CALL JOB:SEARCH-R1-S13D
SET P048 P006
SFTON3D P048
SMOVL C00288 BC00288 V=166.7  +MOVJ EC00288
MOVL C00289 BC00289 V=1000.0  +MOVJ EC00289 VJ=100.00
'EndPath S4334
'Path S4335
SFTOF3D
MOVJ C00290 BC00290 VJ=100.00  +MOVJ EC00290 VJ=100.00
MOVL C00291 BC00291 V=800.0  +MOVJ EC00291 VJ=100.00
SMOVL C00292 BC00292 V=166.7  +MOVJ EC00292
SREFP 3 C00293 BC00293  +REFP EC00293
CALL JOB:SEARCH-R1-S13D
SET P047 P006
SFTON3D P047
SMOVL C00294 BC00294 V=250.0  +MOVJ EC00294
SMOVL C00295 BC00295 V=166.7  +MOVJ EC00295
SREFP 3 C00296 BC00296  +REFP EC00296
CALL JOB:SEARCH-R1-S13D
SET P047 P006
SFTON3D P047
SMOVL C00297 BC00297 V=166.7  +MOVJ EC00297
MOVL C00298 BC00298 V=1000.0  +MOVJ EC00298 VJ=100.00
'EndPath S4335
MOVJ C00299 BC00299 VJ=100.00  +MOVJ EC00299 VJ=100.00
MOVJ C00300 BC00300 VJ=100.00  +MOVJ EC00300 VJ=100.00
MOVJ C00301 BC00301 VJ=100.00  +MOVJ EC00301 VJ=100.00
MOVJ C00302 BC00302 VJ=100.00  +MOVJ EC00302 VJ=100.00
'Path S4336
SFTOF3D
MOVJ C00303 BC00303 VJ=50.00  +MOVJ EC00303 VJ=50.00
MOVJ C00304 BC00304 VJ=100.00  +MOVJ EC00304 VJ=100.00
MOVL C00305 BC00305 V=800.0  +MOVJ EC00305 VJ=100.00
SMOVL C00306 BC00306 V=166.7  +MOVJ EC00306
SREFP 3 C00307 BC00307  +REFP EC00307
CALL JOB:SEARCH-R1-S13D
SET P046 P006
SFTON3D P046
SMOVL C00308 BC00308 V=250.0  +MOVJ EC00308
SMOVL C00309 BC00309 V=166.7  +MOVJ EC00309
SREFP 3 C00310 BC00310  +REFP EC00310
CALL JOB:SEARCH-R1-S13D
SET P046 P006
SFTON3D P046
SMOVL C00311 BC00311 V=166.7  +MOVJ EC00311
MOVL C00312 BC00312 V=1000.0  +MOVJ EC00312 VJ=100.00
'EndPath S4336
'Path S4337
SFTOF3D
MOVJ C00313 BC00313 VJ=100.00  +MOVJ EC00313 VJ=100.00
MOVL C00314 BC00314 V=800.0  +MOVJ EC00314 VJ=100.00
SMOVL C00315 BC00315 V=166.7  +MOVJ EC00315
SREFP 3 C00316 BC00316  +REFP EC00316
CALL JOB:SEARCH-R1-S13D
SET P050 P006
SFTON3D P050
SMOVL C00317 BC00317 V=166.7  +MOVJ EC00317
SREFP 3 C00318 BC00318  +REFP EC00318
CALL JOB:SEARCH-R1-S13D
SET P050 P006
SFTON3D P050
SMOVL C00319 BC00319 V=166.7  +MOVJ EC00319
MOVL C00320 BC00320 V=1000.0  +MOVJ EC00320 VJ=100.00
'EndPath S4337
'Path S4338
SFTOF3D
MOVJ C00321 BC00321 VJ=100.00  +MOVJ EC00321 VJ=100.00
MOVL C00322 BC00322 V=666.7  +MOVJ EC00322 VJ=100.00
SMOVL C00323 BC00323 V=166.7  +MOVJ EC00323
SREFP 3 C00324 BC00324  +REFP EC00324
CALL JOB:SEARCH-R1-S13D
SET P051 P006
SFTON3D P051
SMOVL C00325 BC00325 V=166.7  +MOVJ EC00325
SREFP 3 C00326 BC00326  +REFP EC00326
CALL JOB:SEARCH-R1-S13D
SET P051 P006
SFTON3D P051
SMOVL C00327 BC00327 V=166.7  +MOVJ EC00327
SMOVL C00328 BC00328 V=166.7  +MOVJ EC00328
SMOVL C00329 BC00329 V=133.3  +MOVJ EC00329
SREFP 3 C00330 BC00330  +REFP EC00330
CALL JOB:SEARCH-R1-S13D
SET P051 P006
SFTON3D P051
SMOVL C00331 BC00331 V=250.0  +MOVJ EC00331
SMOVL C00332 BC00332 V=500.0  +MOVJ EC00332
'EndPath S4338
'Path S4339
SFTOF3D
MOVJ C00333 BC00333 VJ=100.00  +MOVJ EC00333 VJ=100.00
MOVL C00334 BC00334 V=800.0  +MOVJ EC00334 VJ=100.00
SMOVL C00335 BC00335 V=166.7  +MOVJ EC00335
SREFP 3 C00336 BC00336  +REFP EC00336
CALL JOB:SEARCH-R1-S13D
SET P045 P006
SFTON3D P045
SMOVL C00337 BC00337 V=250.0  +MOVJ EC00337
SMOVL C00338 BC00338 V=166.7  +MOVJ EC00338
SREFP 3 C00339 BC00339  +REFP EC00339
CALL JOB:SEARCH-R1-S13D
SET P045 P006
SFTON3D P045
SMOVL C00340 BC00340 V=166.7  +MOVJ EC00340
MOVL C00341 BC00341 V=1000.0  +MOVJ EC00341 VJ=100.00
'EndPath S4339
'Path S4340
SFTOF3D
MOVJ C00342 BC00342 VJ=100.00  +MOVJ EC00342 VJ=100.00
MOVL C00343 BC00343 V=800.0  +MOVJ EC00343 VJ=100.00
SMOVL C00344 BC00344 V=166.7  +MOVJ EC00344
SREFP 3 C00345 BC00345  +REFP EC00345
CALL JOB:SEARCH-R1-S13D
SET P044 P006
SFTON3D P044
SMOVL C00346 BC00346 V=250.0  +MOVJ EC00346
SMOVL C00347 BC00347 V=166.7  +MOVJ EC00347
SREFP 3 C00348 BC00348  +REFP EC00348
CALL JOB:SEARCH-R1-S13D
SET P044 P006
SFTON3D P044
SMOVL C00349 BC00349 V=166.7  +MOVJ EC00349
MOVL C00350 BC00350 V=1000.0  +MOVJ EC00350 VJ=100.00
'EndPath S4340
'Path S4341
SFTOF3D
MOVJ C00351 BC00351 VJ=100.00  +MOVJ EC00351 VJ=100.00
MOVL C00352 BC00352 V=800.0  +MOVJ EC00352 VJ=100.00
SMOVL C00353 BC00353 V=166.7  +MOVJ EC00353
SREFP 3 C00354 BC00354  +REFP EC00354
CALL JOB:SEARCH-R1-S13D
SET P049 P006
SFTON3D P049
SMOVL C00355 BC00355 V=166.7  +MOVJ EC00355
SMOVL C00356 BC00356 V=166.7  +MOVJ EC00356
SREFP 3 C00357 BC00357  +REFP EC00357
CALL JOB:SEARCH-R1-S13D
SET P049 P006
SFTON3D P049
SMOVL C00358 BC00358 V=166.7  +MOVJ EC00358
MOVL C00359 BC00359 V=1000.0  +MOVJ EC00359 VJ=100.00
'EndPath S4341
MOVJ C00360 BC00360 VJ=100.00  +MOVJ EC00360 VJ=100.00
MOVJ C00361 BC00361 VJ=100.00  +MOVJ EC00361 VJ=100.00
'Path S4342
SFTOF3D
MOVJ C00362 BC00362 VJ=100.00  +MOVJ EC00362 VJ=100.00
MOVL C00363 BC00363 V=800.0  +MOVJ EC00363 VJ=100.00
SMOVL C00364 BC00364 V=166.7  +MOVJ EC00364
SREFP 3 C00365 BC00365  +REFP EC00365
CALL JOB:SEARCH-R1-S13D
SET P043 P006
SFTON3D P043
SMOVL C00366 BC00366 V=166.7  +MOVJ EC00366
SMOVL C00367 BC00367 V=166.7  +MOVJ EC00367
SREFP 3 C00368 BC00368  +REFP EC00368
CALL JOB:SEARCH-R1-S13D
SET P043 P006
SFTON3D P043
SMOVL C00369 BC00369 V=166.7  +MOVJ EC00369
MOVL C00370 BC00370 V=1000.0  +MOVJ EC00370 VJ=100.00
'EndPath S4342
'Path S4343
SFTOF3D
MOVJ C00371 BC00371 VJ=100.00  +MOVJ EC00371 VJ=100.00
MOVL C00372 BC00372 V=800.0  +MOVJ EC00372 VJ=100.00
SMOVL C00373 BC00373 V=166.7  +MOVJ EC00373
SREFP 3 C00374 BC00374  +REFP EC00374
CALL JOB:SEARCH-R1-S13D
SET P042 P006
SFTON3D P042
SMOVL C00375 BC00375 V=250.0  +MOVJ EC00375
SMOVL C00376 BC00376 V=166.7  +MOVJ EC00376
SREFP 3 C00377 BC00377  +REFP EC00377
CALL JOB:SEARCH-R1-S13D
SET P042 P006
SFTON3D P042
SMOVL C00378 BC00378 V=166.7  +MOVJ EC00378
MOVL C00379 BC00379 V=1000.0  +MOVJ EC00379 VJ=100.00
'EndPath S4343
MOVJ C00380 BC00380 VJ=100.00  +MOVJ EC00380 VJ=100.00
'
'Path W4344
SFTOF3D
SFTON3D P051
MOVJ C00381 BC00381 VJ=60.00  +MOVJ EC00381 VJ=20.00
SMOVL C00382 BC00382 V=500.0  +MOVJ EC00382
SMOVL C00383 BC00383 V=166.7 PL=0  +MOVJ EC00383
MACRO1 MJ#(0) ARGF14
ARCON
SMOVL C00384 BC00384 V=8.3  +MOVJ EC00384
ARCOF
SMOVL C00385 BC00385 V=800.0  +MOVJ EC00385
SMOVL C00386 BC00386 V=150.0  +MOVJ EC00386
ARCON
SMOVL C00387 BC00387 V=11.7  +MOVJ EC00387
ARCOF
SMOVL C00388 BC00388 V=250.0  +MOVJ EC00388
SMOVL C00389 BC00389 V=500.0  +MOVJ EC00389
SMOVL C00390 BC00390 V=1000.0  +MOVJ EC00390
SFTOF3D
'EndPath W4344
'Path W4345
SFTOF3D
SFTON3D P045
MOVJ C00391 BC00391 VJ=100.00  +MOVJ EC00391 VJ=100.00
SMOVL C00392 BC00392 V=800.0  +MOVJ EC00392
SMOVL C00393 BC00393 V=150.0 PL=0  +MOVJ EC00393
MACRO1 MJ#(0) ARGF21
ARCON
SMOVL C00394 BC00394 V=11.7  +MOVJ EC00394
ARCOF
SMOVL C00395 BC00395 V=800.0  +MOVJ EC00395
SMOVL C00396 BC00396 V=1000.0  +MOVJ EC00396
SFTOF3D
'EndPath W4345
'Path W4346
SFTOF3D
SFTON3D P045
MOVJ C00397 BC00397 VJ=100.00  +MOVJ EC00397 VJ=100.00
SMOVL C00398 BC00398 V=800.0  +MOVJ EC00398
SMOVL C00399 BC00399 V=150.0 PL=0  +MOVJ EC00399
ARCON
SMOVL C00400 BC00400 V=11.7  +MOVJ EC00400
ARCOF
SMOVL C00401 BC00401 V=800.0  +MOVJ EC00401
SMOVL C00402 BC00402 V=1000.0  +MOVJ EC00402
SFTOF3D
'EndPath W4346
'Path W4347
SFTOF3D
SFTON3D P049
MOVJ C00403 BC00403 VJ=100.00  +MOVJ EC00403 VJ=100.00
SMOVL C00404 BC00404 V=800.0  +MOVJ EC00404
SMOVL C00405 BC00405 V=150.0 PL=0  +MOVJ EC00405
ARCON
SMOVL C00406 BC00406 V=11.7  +MOVJ EC00406
ARCOF
SMOVL C00407 BC00407 V=800.0  +MOVJ EC00407
SMOVL C00408 BC00408 V=1000.0  +MOVJ EC00408
SFTOF3D
'EndPath W4347
'Path W4348
SFTOF3D
SFTON3D P050
MOVJ C00409 BC00409 VJ=100.00  +MOVJ EC00409 VJ=100.00
SMOVL C00410 BC00410 V=800.0  +MOVJ EC00410
SMOVL C00411 BC00411 V=150.0 PL=0  +MOVJ EC00411
ARCON
SMOVL C00412 BC00412 V=11.7  +MOVJ EC00412
ARCOF
SMOVL C00413 BC00413 V=800.0  +MOVJ EC00413
SMOVL C00414 BC00414 V=1000.0  +MOVJ EC00414
SFTOF3D
'EndPath W4348
MOVJ C00415 BC00415 VJ=100.00  +MOVJ EC00415 VJ=100.00
MOVJ C00416 BC00416 VJ=100.00  +MOVJ EC00416 VJ=100.00
'1
'uwaga na podajnik
'Path W4349
SFTOF3D
SFTON3D P048
MOVJ C00417 BC00417 VJ=100.00  +MOVJ EC00417 VJ=100.00
SMOVL C00418 BC00418 V=800.0  +MOVJ EC00418
SMOVL C00419 BC00419 V=150.0 PL=0  +MOVJ EC00419
ARCON
SMOVL C00420 BC00420 V=11.7  +MOVJ EC00420
ARCOF
SMOVL C00421 BC00421 V=800.0  +MOVJ EC00421
SMOVL C00422 BC00422 V=1000.0  +MOVJ EC00422
SFTOF3D
'EndPath W4349
'Path W4350
SFTOF3D
SFTON3D P048
MOVJ C00423 BC00423 VJ=100.00  +MOVJ EC00423 VJ=100.00
SMOVL C00424 BC00424 V=800.0  +MOVJ EC00424
SMOVL C00425 BC00425 V=150.0 PL=0  +MOVJ EC00425
ARCON
SMOVL C00426 BC00426 V=11.7  +MOVJ EC00426
ARCOF
SMOVL C00427 BC00427 V=800.0  +MOVJ EC00427
SMOVL C00428 BC00428 V=1000.0  +MOVJ EC00428
SFTOF3D
'EndPath W4350
'Path W4351
SFTOF3D
SFTON3D P047
MOVJ C00429 BC00429 VJ=100.00  +MOVJ EC00429 VJ=100.00
SMOVL C00430 BC00430 V=800.0  +MOVJ EC00430
SMOVL C00431 BC00431 V=150.0 PL=0  +MOVJ EC00431
ARCON
SMOVL C00432 BC00432 V=11.7  +MOVJ EC00432
ARCOF
SMOVL C00433 BC00433 V=800.0  +MOVJ EC00433
SMOVL C00434 BC00434 V=1000.0  +MOVJ EC00434
SFTOF3D
'EndPath W4351
'2
MOVJ C00435 BC00435 VJ=100.00  +MOVJ EC00435 VJ=100.00
MOVJ C00436 BC00436 VJ=100.00  +MOVJ EC00436 VJ=100.00
'Path W4352
SFTOF3D
SFTON3D P043
MOVJ C00437 BC00437 VJ=100.00  +MOVJ EC00437 VJ=100.00
SMOVL C00438 BC00438 V=800.0  +MOVJ EC00438
SMOVL C00439 BC00439 V=150.0 PL=0  +MOVJ EC00439
ARCON
SMOVL C00440 BC00440 V=11.7  +MOVJ EC00440
ARCOF
SMOVL C00441 BC00441 V=800.0  +MOVJ EC00441
SMOVL C00442 BC00442 V=1000.0  +MOVJ EC00442
SFTOF3D
'EndPath W4352
'Path W4353
SFTOF3D
SFTON3D P043
MOVJ C00443 BC00443 VJ=100.00  +MOVJ EC00443 VJ=100.00
SMOVL C00444 BC00444 V=800.0  +MOVJ EC00444
SMOVL C00445 BC00445 V=150.0 PL=0  +MOVJ EC00445
ARCON
SMOVL C00446 BC00446 V=11.7  +MOVJ EC00446
ARCOF
SMOVL C00447 BC00447 V=800.0  +MOVJ EC00447
SMOVL C00448 BC00448 V=1000.0  +MOVJ EC00448
SFTOF3D
'EndPath W4353
'Path W4354
SFTOF3D
SFTON3D P042
MOVJ C00449 BC00449 VJ=100.00  +MOVJ EC00449 VJ=100.00
SMOVL C00450 BC00450 V=800.0  +MOVJ EC00450
SMOVL C00451 BC00451 V=150.0 PL=0  +MOVJ EC00451
ARCON
SMOVL C00452 BC00452 V=11.7  +MOVJ EC00452
ARCOF
SMOVL C00453 BC00453 V=800.0  +MOVJ EC00453
SMOVL C00454 BC00454 V=1000.0  +MOVJ EC00454
SFTOF3D
'EndPath W4354
'Path W4355
SFTOF3D
SFTON3D P042
MOVJ C00455 BC00455 VJ=100.00  +MOVJ EC00455 VJ=100.00
SMOVL C00456 BC00456 V=800.0  +MOVJ EC00456
SMOVL C00457 BC00457 V=150.0 PL=0  +MOVJ EC00457
ARCON
SMOVL C00458 BC00458 V=11.7  +MOVJ EC00458
ARCOF
SMOVL C00459 BC00459 V=800.0  +MOVJ EC00459
SMOVL C00460 BC00460 V=1000.0  +MOVJ EC00460
SFTOF3D
'EndPath W4355
'3
MOVJ C00461 BC00461 VJ=100.00  +MOVJ EC00461 VJ=100.00
'Path W4356
SFTOF3D
SFTON3D P044
MOVJ C00462 BC00462 VJ=100.00  +MOVJ EC00462 VJ=100.00
SMOVL C00463 BC00463 V=800.0  +MOVJ EC00463
SMOVL C00464 BC00464 V=150.0 PL=0  +MOVJ EC00464
ARCON
SMOVL C00465 BC00465 V=11.7  +MOVJ EC00465
ARCOF
SMOVL C00466 BC00466 V=800.0  +MOVJ EC00466
SMOVL C00467 BC00467 V=1000.0  +MOVJ EC00467
SFTOF3D
'EndPath W4356
'Path W4357
SFTOF3D
SFTON3D P046
MOVJ C00468 BC00468 VJ=100.00  +MOVJ EC00468 VJ=100.00
SMOVL C00469 BC00469 V=800.0  +MOVJ EC00469
SMOVL C00470 BC00470 V=150.0 PL=0  +MOVJ EC00470
MACRO1 MJ#(0) ARGF14
ARCON
SMOVL C00471 BC00471 V=11.7  +MOVJ EC00471
ARCOF
SMOVL C00472 BC00472 V=800.0  +MOVJ EC00472
SMOVL C00473 BC00473 V=1000.0  +MOVJ EC00473
SFTOF3D
'EndPath W4357
MOVJ C00474 BC00474 VJ=100.00  +MOVJ EC00474 VJ=100.00
MOVJ C00475 BC00475 VJ=100.00  +MOVJ EC00475 VJ=100.00
MOVJ C00476 BC00476 VJ=100.00  +MOVJ EC00476 VJ=100.00
END
